LIN {X 0,Y 167.606,Z 477.864,A -85,B 0,C 180,E1 -23684.106,E2 -23684.106} C_VEL
LIN {X 0,Y 165.096,Z 487.968,A -85,B 0,C 180,E1 -23686.634,E2 -23686.634} C_VEL
LIN {X 0,Y 162.293,Z 498.184,A -85,B 0,C 180,E1 -23689.862,E2 -23689.862} C_VEL
LIN {X 0,Y 159.942,Z 506.695,A -85,B 0,C 180,E1 -23693.294,E2 -23693.294} C_VEL
LIN {X 0,Y 157.877,Z 514.165,A -85,B 0,C 180,E1 -23697.088,E2 -23697.088} C_VEL
LIN {X 0,Y 156.257,Z 520.604,A -85,B 0,C 180,E1 -23701.288,E2 -23701.288} C_VEL
LIN {X 0,Y 155.089,Z 526.085,A -85,B 0,C 180,E1 -23706.092,E2 -23706.092} C_VEL
LIN {X 0,Y 154.517,Z 529.018,A -85,B 0,C 180,E1 -23709.55,E2 -23709.55} C_VEL
LIN {X 0,Y 154.343,Z 531.312,A -85,B 0,C 180,E1 -23713.234,E2 -23713.234} C_VEL
LIN {X 0,Y 154.636,Z 532.81,A -85,B 0,C 180,E1 -23717.021,E2 -23717.021} C_VEL
LIN {X 0,Y 155.395,Z 533.466,A -85,B 0,C 180,E1 -23720.715,E2 -23720.715} C_VEL
LIN {X 0,Y 156.609,Z 533.371,A -85,B 0,C 180,E1 -23724.311,E2 -23724.311} C_VEL
LIN {X 0,Y 158.291,Z 532.569,A -85,B 0,C 180,E1 -23727.806,E2 -23727.806} C_VEL
LIN {X 0,Y 161.621,Z 529.982,A -85,B 0,C 180,E1 -23732.838,E2 -23732.838} C_VEL
LIN {X 0,Y 166.003,Z 525.79,A -85,B 0,C 180,E1 -23737.603,E2 -23737.603} C_VEL
LIN {X 0,Y 170.548,Z 520.782,A -85,B 0,C 180,E1 -23741.4,E2 -23741.4} C_VEL
LIN {X 0,Y 175.041,Z 515.343,A -85,B 0,C 180,E1 -23744.491,E2 -23744.491} C_VEL
LIN {X 0,Y 180.004,Z 508.62,A -85,B 0,C 180,E1 -23747.439,E2 -23747.439} C_VEL
LIN {X 0,Y 185.416,Z 500.371,A -85,B 0,C 180,E1 -23750.225,E2 -23750.225} C_VEL
LIN {X 0,Y 185.994,Z 499.153,A -85,B 0,C 180,E1 -23750.652,E2 -23750.652} C_VEL
LIN {X 0,Y 186.922,Z 493.836,A -85,B 0,C 180,E1 -23752.981,E2 -23752.981} C_VEL
LIN {X 0,Y 187.381,Z 487.918,A -85,B 0,C 180,E1 -23755.698,E2 -23755.698} C_VEL
LIN {X 0,Y 187.227,Z 483.523,A -85,B 0,C 180,E1 -23757.849,E2 -23757.849} C_VEL
LIN {X 0,Y 185.998,Z 477.859,A -85,B 0,C 180,E1 -23761.323,E2 -23761.323} C_VEL
LIN {X 0,Y 184.814,Z 473.591,A -85,B 0,C 180,E1 -23764.362,E2 -23764.362} C_VEL
LIN {X 0,Y 182.814,Z 469.179,A -85,B 0,C 180,E1 -23768.846,E2 -23768.846} C_VEL
LIN {X 0,Y 181.491,Z 465.804,A -85,B 0,C 180,E1 -23773.435,E2 -23773.435} C_VEL
LIN {X 0,Y 180.179,Z 465.166,A -85,B 0,C 180,E1 -23778.183,E2 -23778.183} C_VEL
LIN {X 0,Y 179.96,Z 465.653,A -85,B 0,C 180,E1 -23782.988,E2 -23782.988} C_VEL
LIN {X 0,Y 180.833,Z 467.315,A -85,B 0,C 180,E1 -23787.8,E2 -23787.8} C_VEL
LIN {X 0,Y 181.658,Z 470.723,A -85,B 0,C 180,E1 -23791.667,E2 -23791.667} C_VEL
LIN {X 0,Y 183.014,Z 474.33,A -85,B 0,C 180,E1 -23795.172,E2 -23795.172} C_VEL
LIN {X 0,Y 184.207,Z 478.675,A -85,B 0,C 180,E1 -23798.299,E2 -23798.299} C_VEL
LIN {X 0,Y 185.126,Z 482.365,A -85,B 0,C 180,E1 -23800.602,E2 -23800.602} C_VEL
LIN {X 0,Y 186.038,Z 487.75,A -85,B 0,C 180,E1 -23803.498,E2 -23803.498} C_VEL
LIN {X 0,Y 186.059,Z 492.37,A -85,B 0,C 180,E1 -23805.496,E2 -23805.496} C_VEL
LIN {X 0,Y 184.829,Z 499.849,A -85,B 0,C 180,E1 -23808.287,E2 -23808.287} C_VEL
LIN {X 0,Y 182.79,Z 507.719,A -85,B 0,C 180,E1 -23811.262,E2 -23811.262} C_VEL
LIN {X 0,Y 180.399,Z 513.668,A -85,B 0,C 180,E1 -23813.552,E2 -23813.552} C_VEL
LIN {X 0,Y 175.085,Z 521.477,A -85,B 0,C 180,E1 -23816.502,E2 -23816.502} C_VEL
LIN {X 0,Y 169.515,Z 528.822,A -85,B 0,C 180,E1 -23820.166,E2 -23820.166} C_VEL
LIN {X 0,Y 165.518,Z 533.839,A -85,B 0,C 180,E1 -23823.524,E2 -23823.524} C_VEL
LIN {X 0,Y 161.075,Z 538.896,A -85,B 0,C 180,E1 -23828.232,E2 -23828.232} C_VEL
LIN {X 0,Y 158.362,Z 541.598,A -85,B 0,C 180,E1 -23831.902,E2 -23831.902} C_VEL
LIN {X 0,Y 156.117,Z 543.873,A -85,B 0,C 180,E1 -23836.993,E2 -23836.993} C_VEL
LIN {X 0,Y 154.964,Z 544.594,A -85,B 0,C 180,E1 -23842.181,E2 -23842.181} C_VEL
LIN {X 0,Y 154.845,Z 543.82,A -85,B 0,C 180,E1 -23847.4,E2 -23847.4} C_VEL
LIN {X 0,Y 155.038,Z 542.857,A -85,B 0,C 180,E1 -23850.001,E2 -23850.001} C_VEL
LIN {X 0,Y 154.859,Z 541.002,A -85,B 0,C 180,E1 -23853.207,E2 -23853.207} C_VEL
LIN {X 0,Y 155.118,Z 537.201,A -85,B 0,C 180,E1 -23857.813,E2 -23857.813} C_VEL
LIN {X 0,Y 155.754,Z 532.742,A -85,B 0,C 180,E1 -23861.716,E2 -23861.716} C_VEL
LIN {X 0,Y 157.161,Z 525.927,A -85,B 0,C 180,E1 -23866.231,E2 -23866.231} C_VEL
LIN {X 0,Y 159.131,Z 518.527,A -85,B 0,C 180,E1 -23870.017,E2 -23870.017} C_VEL
LIN {X 0,Y 161.442,Z 509.83,A -85,B 0,C 180,E1 -23873.536,E2 -23873.536} C_VEL
LIN {X 0,Y 164.242,Z 499.771,A -85,B 0,C 180,E1 -23876.7,E2 -23876.7} C_VEL
LIN {X 0,Y 164.795,Z 496.433,A -85,B 0,C 180,E1 -23877.633,E2 -23877.633} C_VEL
LIN {X 0,Y 164.825,Z 485.619,A -85,B 0,C 180,E1 -23880.421,E2 -23880.421} C_VEL
LIN {X 0,Y 164.622,Z 480.666,A -85,B 0,C 180,E1 -23881.556,E2 -23881.556} C_VEL
LIN {X 0,Y 163.709,Z 475.807,A -85,B 0,C 180,E1 -23882.687,E2 -23882.687} C_VEL
LIN {X 0,Y 160.346,Z 468.173,A -85,B 0,C 180,E1 -23884.594,E2 -23884.594} C_VEL
LIN {X 0,Y 156.75,Z 460.325,A -85,B 0,C 180,E1 -23886.407,E2 -23886.407} C_VEL
LIN {X 0,Y 155.458,Z 455.118,A -85,B 0,C 180,E1 -23887.351,E2 -23887.351} C_VEL
LIN {X 0,Y 153.531,Z 445.023,A -85,B 0,C 180,E1 -23888.904,E2 -23888.904} C_VEL
LIN {X 0,Y 151.69,Z 438.84,A -85,B 0,C 180,E1 -23889.901,E2 -23889.901} C_VEL
LIN {X 0,Y 150.938,Z 435.132,A -85,B 0,C 180,E1 -23895.698,E2 -23895.698} C_VEL
LIN {X 0,Y 150.396,Z 431.753,A -85,B 0,C 180,E1 -23901.316,E2 -23901.316} C_VEL
LIN {X 0,Y 150.224,Z 431.776,A -85,B 0,C 180,E1 -23907.364,E2 -23907.364} C_VEL
LIN {X 0,Y 150.247,Z 431.754,A -85,B 0,C 180,E1 -23912.718,E2 -23912.718} C_VEL
LIN {X 0,Y 150.354,Z 431.756,A -85,B 0,C 180,E1 -23919.208,E2 -23919.208} C_VEL
LIN {X 0,Y 150.385,Z 431.751,A -85,B 0,C 180,E1 -23923.716,E2 -23923.716} C_VEL
LIN {X 0,Y 150.661,Z 431.712,A -85,B 0,C 180,E1 -23929.246,E2 -23929.246} C_VEL
LIN {X 0,Y 150.747,Z 431.705,A -85,B 0,C 180,E1 -23931.96,E2 -23931.96} C_VEL
LIN {X 0,Y 151.219,Z 431.645,A -85,B 0,C 180,E1 -23940,E2 -23940} C_VEL
LIN {X 0,Y 150.747,Z 431.703,A -85,B 0,C 180,E1 -23948.04,E2 -23948.04} C_VEL
LIN {X 0,Y 150.616,Z 431.717,A -85,B 0,C 180,E1 -23951.506,E2 -23951.506} C_VEL
LIN {X 0,Y 150.369,Z 431.724,A -85,B 0,C 180,E1 -23956.286,E2 -23956.286} C_VEL
LIN {X 0,Y 150.353,Z 431.734,A -85,B 0,C 180,E1 -23960.792,E2 -23960.792} C_VEL
LIN {X 0,Y 150.247,Z 431.769,A -85,B 0,C 180,E1 -23967.282,E2 -23967.282} C_VEL
LIN {X 0,Y 150.217,Z 431.757,A -85,B 0,C 180,E1 -23972.632,E2 -23972.632} C_VEL
LIN {X 0,Y 150.174,Z 431.754,A -85,B 0,C 180,E1 -23977.473,E2 -23977.473} C_VEL
LIN {X 0,Y 150.138,Z 431.779,A -85,B 0,C 180,E1 -23981.498,E2 -23981.498} C_VEL
LIN {X 0,Y 150.127,Z 431.782,A -85,B 0,C 180,E1 -23985.395,E2 -23985.395} C_VEL
LIN {X 0,Y 150.157,Z 431.764,A -85,B 0,C 180,E1 -23989.06,E2 -23989.06} C_VEL
LIN {X 0,Y 150.217,Z 431.756,A -85,B 0,C 180,E1 -23992.689,E2 -23992.689} C_VEL
LIN {X 0,Y 150.221,Z 431.772,A -85,B 0,C 180,E1 -23997.365,E2 -23997.365} C_VEL
LIN {X 0,Y 150.246,Z 431.755,A -85,B 0,C 180,E1 -24002.717,E2 -24002.717} C_VEL
LIN {X 0,Y 150.353,Z 431.755,A -85,B 0,C 180,E1 -24009.207,E2 -24009.207} C_VEL
LIN {X 0,Y 150.385,Z 431.75,A -85,B 0,C 180,E1 -24013.715,E2 -24013.715} C_VEL
LIN {X 0,Y 150.691,Z 431.709,A -85,B 0,C 180,E1 -24019.247,E2 -24019.247} C_VEL
LIN {X 0,Y 150.765,Z 431.706,A -85,B 0,C 180,E1 -24021.96,E2 -24021.96} C_VEL
LIN {X 0,Y 151.21,Z 431.654,A -85,B 0,C 180,E1 -24029.999,E2 -24029.999} C_VEL
LIN {X 0,Y 150.747,Z 431.7,A -85,B 0,C 180,E1 -24033.34,E2 -24033.34} C_VEL
LIN {X 0,Y 151.68,Z 434.542,A -85,B 0,C 180,E1 -24033.818,E2 -24033.818} C_VEL
LIN {X 0,Y 155.095,Z 443.394,A -85,B 0,C 180,E1 -24035.557,E2 -24035.557} C_VEL
LIN {X 0,Y 157.769,Z 455.58,A -85,B 0,C 180,E1 -24037.913,E2 -24037.913} C_VEL
LIN {X 0,Y 159.591,Z 466.873,A -85,B 0,C 180,E1 -24040.404,E2 -24040.404} C_VEL
LIN {X 0,Y 160.717,Z 477.996,A -85,B 0,C 180,E1 -24043.238,E2 -24043.238} C_VEL
LIN {X 0,Y 160.38,Z 480.569,A -85,B 0,C 180,E1 -24043.879,E2 -24043.879} C_VEL
LIN {X 0,Y 157.438,Z 491.337,A -85,B 0,C 180,E1 -24046.866,E2 -24046.866} C_VEL
LIN {X 0,Y 154.862,Z 500.222,A -85,B 0,C 180,E1 -24049.976,E2 -24049.976} C_VEL
LIN {X 0,Y 152.388,Z 508.801,A -85,B 0,C 180,E1 -24053.751,E2 -24053.751} C_VEL
LIN {X 0,Y 150.329,Z 516.089,A -85,B 0,C 180,E1 -24057.871,E2 -24057.871} C_VEL
LIN {X 0,Y 148.934,Z 521.626,A -85,B 0,C 180,E1 -24061.854,E2 -24061.854} C_VEL
LIN {X 0,Y 147.962,Z 526.248,A -85,B 0,C 180,E1 -24066.15,E2 -24066.15} C_VEL
LIN {X 0,Y 147.347,Z 529.542,A -85,B 0,C 180,E1 -24070.257,E2 -24070.257} C_VEL
LIN {X 0,Y 147.363,Z 532.428,A -85,B 0,C 180,E1 -24075.672,E2 -24075.672} C_VEL
LIN {X 0,Y 147.951,Z 533.48,A -85,B 0,C 180,E1 -24079.465,E2 -24079.465} C_VEL
LIN {X 0,Y 149.059,Z 533.812,A -85,B 0,C 180,E1 -24083.275,E2 -24083.275} C_VEL
LIN {X 0,Y 150.696,Z 533.398,A -85,B 0,C 180,E1 -24087.081,E2 -24087.081} C_VEL
LIN {X 0,Y 152.883,Z 532.17,A -85,B 0,C 180,E1 -24090.856,E2 -24090.856} C_VEL
LIN {X 0,Y 155.665,Z 530.091,A -85,B 0,C 180,E1 -24094.547,E2 -24094.547} C_VEL
LIN {X 0,Y 160.591,Z 525.711,A -85,B 0,C 180,E1 -24099.506,E2 -24099.506} C_VEL
LIN {X 0,Y 164.468,Z 521.812,A -85,B 0,C 180,E1 -24102.595,E2 -24102.595} C_VEL
LIN {X 0,Y 169.809,Z 515.754,A -85,B 0,C 180,E1 -24106.161,E2 -24106.161} C_VEL
LIN {X 0,Y 175.977,Z 507.825,A -85,B 0,C 180,E1 -24109.608,E2 -24109.608} C_VEL
LIN {X 0,Y 180.019,Z 502.001,A -85,B 0,C 180,E1 -24111.582,E2 -24111.582} C_VEL
LIN {X 0,Y 181.132,Z 498.231,A -85,B 0,C 180,E1 -24113.316,E2 -24113.316} C_VEL
LIN {X 0,Y 182.048,Z 491.436,A -85,B 0,C 180,E1 -24116.68,E2 -24116.68} C_VEL
LIN {X 0,Y 182.083,Z 487.42,A -85,B 0,C 180,E1 -24118.894,E2 -24118.894} C_VEL
LIN {X 0,Y 181.269,Z 482.422,A -85,B 0,C 180,E1 -24122.222,E2 -24122.222} C_VEL
LIN {X 0,Y 180.702,Z 479.514,A -85,B 0,C 180,E1 -24124.461,E2 -24124.461} C_VEL
LIN {X 0,Y 179.095,Z 475.199,A -85,B 0,C 180,E1 -24129.031,E2 -24129.031} C_VEL
LIN {X 0,Y 178.032,Z 471.992,A -85,B 0,C 180,E1 -24133.701,E2 -24133.701} C_VEL
LIN {X 0,Y 176.861,Z 471.49,A -85,B 0,C 180,E1 -24138.536,E2 -24138.536} C_VEL
LIN {X 0,Y 176.759,Z 472.209,A -85,B 0,C 180,E1 -24143.87,E2 -24143.87} C_VEL
LIN {X 0,Y 177.032,Z 472.822,A -85,B 0,C 180,E1 -24145.893,E2 -24145.893} C_VEL
LIN {X 0,Y 177.487,Z 474.141,A -85,B 0,C 180,E1 -24148.37,E2 -24148.37} C_VEL
LIN {X 0,Y 178.9,Z 479.645,A -85,B 0,C 180,E1 -24154.416,E2 -24154.416} C_VEL
LIN {X 0,Y 180.101,Z 485.351,A -85,B 0,C 180,E1 -24158.7,E2 -24158.7} C_VEL
LIN {X 0,Y 180.932,Z 491.56,A -85,B 0,C 180,E1 -24162.439,E2 -24162.439} C_VEL
LIN {X 0,Y 180.932,Z 494.505,A -85,B 0,C 180,E1 -24163.904,E2 -24163.904} C_VEL
LIN {X 0,Y 179.545,Z 501.474,A -85,B 0,C 180,E1 -24166.765,E2 -24166.765} C_VEL
LIN {X 0,Y 177.218,Z 509.076,A -85,B 0,C 180,E1 -24169.852,E2 -24169.852} C_VEL
LIN {X 0,Y 174.751,Z 514.717,A -85,B 0,C 180,E1 -24172.172,E2 -24172.172} C_VEL
LIN {X 0,Y 171.1,Z 519.894,A -85,B 0,C 180,E1 -24174.175,E2 -24174.175} C_VEL
LIN {X 0,Y 164.997,Z 527.506,A -85,B 0,C 180,E1 -24177.831,E2 -24177.831} C_VEL
LIN {X 0,Y 160.529,Z 532.689,A -85,B 0,C 180,E1 -24181.213,E2 -24181.213} C_VEL
LIN {X 0,Y 156.721,Z 536.813,A -85,B 0,C 180,E1 -24184.786,E2 -24184.786} C_VEL
LIN {X 0,Y 153.459,Z 539.994,A -85,B 0,C 180,E1 -24188.509,E2 -24188.509} C_VEL
LIN {X 0,Y 150.183,Z 542.867,A -85,B 0,C 180,E1 -24193.695,E2 -24193.695} C_VEL
LIN {X 0,Y 148.4,Z 544.179,A -85,B 0,C 180,E1 -24199.081,E2 -24199.081} C_VEL
LIN {X 0,Y 147.702,Z 544.023,A -85,B 0,C 180,E1 -24204.54,E2 -24204.54} C_VEL
LIN {X 0,Y 147.756,Z 543.383,A -85,B 0,C 180,E1 -24207.275,E2 -24207.275} C_VEL
LIN {X 0,Y 147.961,Z 542.311,A -85,B 0,C 180,E1 -24210.001,E2 -24210.001} C_VEL
LIN {X 0,Y 147.796,Z 540.593,A -85,B 0,C 180,E1 -24213.033,E2 -24213.033} C_VEL
LIN {X 0,Y 147.941,Z 537.676,A -85,B 0,C 180,E1 -24216.822,E2 -24216.822} C_VEL
LIN {X 0,Y 148.476,Z 533.464,A -85,B 0,C 180,E1 -24220.915,E2 -24220.915} C_VEL
LIN {X 0,Y 149.753,Z 527.028,A -85,B 0,C 180,E1 -24225.656,E2 -24225.656} C_VEL
LIN {X 0,Y 151.698,Z 519.972,A -85,B 0,C 180,E1 -24229.627,E2 -24229.627} C_VEL
LIN {X 0,Y 154.109,Z 511.148,A -85,B 0,C 180,E1 -24233.519,E2 -24233.519} C_VEL
LIN {X 0,Y 157.057,Z 501.178,A -85,B 0,C 180,E1 -24236.942,E2 -24236.942} C_VEL
LIN {X 0,Y 157.864,Z 498.001,A -85,B 0,C 180,E1 -24237.87,E2 -24237.87} C_VEL
LIN {X 0,Y 158.009,Z 487.611,A -85,B 0,C 180,E1 -24240.765,E2 -24240.765} C_VEL
LIN {X 0,Y 157.549,Z 475.881,A -85,B 0,C 180,E1 -24243.507,E2 -24243.507} C_VEL
LIN {X 0,Y 156.47,Z 462.878,A -85,B 0,C 180,E1 -24246.051,E2 -24246.051} C_VEL
LIN {X 0,Y 155.458,Z 455.118,A -85,B 0,C 180,E1 -24247.351,E2 -24247.351} C_VEL
LIN {X 0,Y 154.222,Z 451.815,A -85,B 0,C 180,E1 -24248.012,E2 -24248.012} C_VEL
LIN {X 0,Y 150.308,Z 447.483,A -85,B 0,C 180,E1 -24249.296,E2 -24249.296} C_VEL
LIN {X 0,Y 146.203,Z 443.152,A -85,B 0,C 180,E1 -24250.592,E2 -24250.592} C_VEL
LIN {X 0,Y 144.647,Z 439.82,A -85,B 0,C 180,E1 -24251.226,E2 -24251.226} C_VEL
LIN {X 0,Y 144.416,Z 438.578,A -85,B 0,C 180,E1 -24251.433,E2 -24251.433} C_VEL
LIN {X 0,Y 143.699,Z 435.125,A -85,B 0,C 180,E1 -24257.191,E2 -24257.191} C_VEL
LIN {X 0,Y 143.319,Z 432.633,A -85,B 0,C 180,E1 -24261.685,E2 -24261.685} C_VEL
LIN {X 0,Y 143.191,Z 432.651,A -85,B 0,C 180,E1 -24267.323,E2 -24267.323} C_VEL
LIN {X 0,Y 143.195,Z 432.634,A -85,B 0,C 180,E1 -24272.062,E2 -24272.062} C_VEL
LIN {X 0,Y 143.28,Z 432.639,A -85,B 0,C 180,E1 -24278.746,E2 -24278.746} C_VEL
LIN {X 0,Y 143.319,Z 432.629,A -85,B 0,C 180,E1 -24282.889,E2 -24282.889} C_VEL
LIN {X 0,Y 143.597,Z 432.591,A -85,B 0,C 180,E1 -24288.71,E2 -24288.71} C_VEL
LIN {X 0,Y 143.668,Z 432.588,A -85,B 0,C 180,E1 -24291.561,E2 -24291.561} C_VEL
LIN {X 0,Y 144.178,Z 432.522,A -85,B 0,C 180,E1 -24300,E2 -24300} C_VEL
LIN {X 0,Y 143.668,Z 432.586,A -85,B 0,C 180,E1 -24308.439,E2 -24308.439} C_VEL
LIN {X 0,Y 143.55,Z 432.597,A -85,B 0,C 180,E1 -24311.712,E2 -24311.712} C_VEL
LIN {X 0,Y 143.307,Z 432.597,A -85,B 0,C 180,E1 -24317.112,E2 -24317.112} C_VEL
LIN {X 0,Y 143.279,Z 432.617,A -85,B 0,C 180,E1 -24321.254,E2 -24321.254} C_VEL
LIN {X 0,Y 143.193,Z 432.647,A -85,B 0,C 180,E1 -24327.937,E2 -24327.937} C_VEL
LIN {X 0,Y 143.166,Z 432.631,A -85,B 0,C 180,E1 -24333.432,E2 -24333.432} C_VEL
LIN {X 0,Y 143.057,Z 432.655,A -85,B 0,C 180,E1 -24339.691,E2 -24339.691} C_VEL
LIN {X 0,Y 143.036,Z 432.666,A -85,B 0,C 180,E1 -24343.463,E2 -24343.463} C_VEL
LIN {X 0,Y 143.069,Z 432.655,A -85,B 0,C 180,E1 -24347.464,E2 -24347.464} C_VEL
LIN {X 0,Y 143.108,Z 432.637,A -85,B 0,C 180,E1 -24351.791,E2 -24351.791} C_VEL
LIN {X 0,Y 143.188,Z 432.648,A -85,B 0,C 180,E1 -24357.322,E2 -24357.322} C_VEL
LIN {X 0,Y 143.192,Z 432.635,A -85,B 0,C 180,E1 -24362.062,E2 -24362.062} C_VEL
LIN {X 0,Y 143.279,Z 432.637,A -85,B 0,C 180,E1 -24368.744,E2 -24368.744} C_VEL
LIN {X 0,Y 143.318,Z 432.627,A -85,B 0,C 180,E1 -24372.888,E2 -24372.888} C_VEL
LIN {X 0,Y 143.604,Z 432.592,A -85,B 0,C 180,E1 -24378.71,E2 -24378.71} C_VEL
LIN {X 0,Y 143.686,Z 432.587,A -85,B 0,C 180,E1 -24381.561,E2 -24381.561} C_VEL
LIN {X 0,Y 144.165,Z 432.531,A -85,B 0,C 180,E1 -24389.999,E2 -24389.999} C_VEL
LIN {X 0,Y 143.851,Z 432.562,A -85,B 0,C 180,E1 -24391.924,E2 -24391.924} C_VEL
LIN {X 0,Y 145.748,Z 437.9,A -85,B 0,C 180,E1 -24392.972,E2 -24392.972} C_VEL
LIN {X 0,Y 149.007,Z 446.478,A -85,B 0,C 180,E1 -24394.801,E2 -24394.801} C_VEL
LIN {X 0,Y 151.453,Z 458.476,A -85,B 0,C 180,E1 -24397.33,E2 -24397.33} C_VEL
LIN {X 0,Y 153.11,Z 470.258,A -85,B 0,C 180,E1 -24400.169,E2 -24400.169} C_VEL
LIN {X 0,Y 153.87,Z 480.076,A -85,B 0,C 180,E1 -24402.864,E2 -24402.864} C_VEL
LIN {X 0,Y 150.956,Z 490.342,A -85,B 0,C 180,E1 -24405.735,E2 -24405.735} C_VEL
LIN {X 0,Y 147.914,Z 500.569,A -85,B 0,C 180,E1 -24409.425,E2 -24409.425} C_VEL
LIN {X 0,Y 145.382,Z 508.987,A -85,B 0,C 180,E1 -24413.293,E2 -24413.293} C_VEL
LIN {X 0,Y 143.513,Z 515.375,A -85,B 0,C 180,E1 -24416.988,E2 -24416.988} C_VEL
LIN {X 0,Y 142.076,Z 520.933,A -85,B 0,C 180,E1 -24421.004,E2 -24421.004} C_VEL
LIN {X 0,Y 141.079,Z 525.25,A -85,B 0,C 180,E1 -24424.95,E2 -24424.95} C_VEL
LIN {X 0,Y 140.403,Z 528.463,A -85,B 0,C 180,E1 -24428.73,E2 -24428.73} C_VEL
LIN {X 0,Y 140.182,Z 530.173,A -85,B 0,C 180,E1 -24431.234,E2 -24431.234} C_VEL
LIN {X 0,Y 140.236,Z 532.319,A -85,B 0,C 180,E1 -24435.443,E2 -24435.443} C_VEL
LIN {X 0,Y 140.846,Z 533.611,A -85,B 0,C 180,E1 -24439.558,E2 -24439.558} C_VEL
LIN {X 0,Y 141.999,Z 534.126,A -85,B 0,C 180,E1 -24443.565,E2 -24443.565} C_VEL
LIN {X 0,Y 143.654,Z 533.853,A -85,B 0,C 180,E1 -24447.442,E2 -24447.442} C_VEL
LIN {X 0,Y 145.807,Z 532.885,A -85,B 0,C 180,E1 -24451.183,E2 -24451.183} C_VEL
LIN {X 0,Y 149.992,Z 530.143,A -85,B 0,C 180,E1 -24456.531,E2 -24456.531} C_VEL
LIN {X 0,Y 155.476,Z 525.543,A -85,B 0,C 180,E1 -24461.666,E2 -24461.666} C_VEL
LIN {X 0,Y 161.117,Z 520.115,A -85,B 0,C 180,E1 -24465.693,E2 -24465.693} C_VEL
LIN {X 0,Y 167.273,Z 513.308,A -85,B 0,C 180,E1 -24469.328,E2 -24469.328} C_VEL
LIN {X 0,Y 173.825,Z 504.974,A -85,B 0,C 180,E1 -24472.597,E2 -24472.597} C_VEL
LIN {X 0,Y 174.701,Z 503.68,A -85,B 0,C 180,E1 -24473.068,E2 -24473.068} C_VEL
LIN {X 0,Y 175.951,Z 499.129,A -85,B 0,C 180,E1 -24475.418,E2 -24475.418} C_VEL
LIN {X 0,Y 176.722,Z 494.898,A -85,B 0,C 180,E1 -24477.721,E2 -24477.721} C_VEL
LIN {X 0,Y 176.899,Z 491.184,A -85,B 0,C 180,E1 -24480,E2 -24480} C_VEL
LIN {X 0,Y 176.439,Z 486.58,A -85,B 0,C 180,E1 -24483.426,E2 -24483.426} C_VEL
LIN {X 0,Y 175.934,Z 484.022,A -85,B 0,C 180,E1 -24485.732,E2 -24485.732} C_VEL
LIN {X 0,Y 175.056,Z 481.008,A -85,B 0,C 180,E1 -24489.241,E2 -24489.241} C_VEL
LIN {X 0,Y 174.117,Z 477.936,A -85,B 0,C 180,E1 -24494.372,E2 -24494.372} C_VEL
LIN {X 0,Y 173.055,Z 477.751,A -85,B 0,C 180,E1 -24500.927,E2 -24500.927} C_VEL
LIN {X 0,Y 173.161,Z 478.355,A -85,B 0,C 180,E1 -24503.946,E2 -24503.946} C_VEL
LIN {X 0,Y 173.494,Z 479.509,A -85,B 0,C 180,E1 -24506.98,E2 -24506.98} C_VEL
LIN {X 0,Y 173.848,Z 481.766,A -85,B 0,C 180,E1 -24510.209,E2 -24510.209} C_VEL
LIN {X 0,Y 174.675,Z 485.537,A -85,B 0,C 180,E1 -24514.284,E2 -24514.284} C_VEL
LIN {X 0,Y 175.348,Z 490.022,A -85,B 0,C 180,E1 -24517.874,E2 -24517.874} C_VEL
LIN {X 0,Y 175.754,Z 495.166,A -85,B 0,C 180,E1 -24521.283,E2 -24521.283} C_VEL
LIN {X 0,Y 175.566,Z 498.618,A -85,B 0,C 180,E1 -24523.148,E2 -24523.148} C_VEL
LIN {X 0,Y 173.888,Z 504.629,A -85,B 0,C 180,E1 -24525.814,E2 -24525.814} C_VEL
LIN {X 0,Y 171.214,Z 511.821,A -85,B 0,C 180,E1 -24528.948,E2 -24528.948} C_VEL
LIN {X 0,Y 168.416,Z 517.048,A -85,B 0,C 180,E1 -24531.249,E2 -24531.249} C_VEL
LIN {X 0,Y 162.646,Z 524.098,A -85,B 0,C 180,E1 -24534.316,E2 -24534.316} C_VEL
LIN {X 0,Y 157.393,Z 529.889,A -85,B 0,C 180,E1 -24537.601,E2 -24537.601} C_VEL
LIN {X 0,Y 153.566,Z 533.91,A -85,B 0,C 180,E1 -24540.622,E2 -24540.622} C_VEL
LIN {X 0,Y 149.094,Z 538.173,A -85,B 0,C 180,E1 -24544.899,E2 -24544.899} C_VEL
LIN {X 0,Y 144.922,Z 541.632,A -85,B 0,C 180,E1 -24550.157,E2 -24550.157} C_VEL
LIN {X 0,Y 142.241,Z 543.529,A -85,B 0,C 180,E1 -24555.698,E2 -24555.698} C_VEL
LIN {X 0,Y 140.895,Z 543.974,A -85,B 0,C 180,E1 -24561.395,E2 -24561.395} C_VEL
LIN {X 0,Y 140.629,Z 543.635,A -85,B 0,C 180,E1 -24564.265,E2 -24564.265} C_VEL
LIN {X 0,Y 140.705,Z 542.799,A -85,B 0,C 180,E1 -24567.404,E2 -24567.404} C_VEL
LIN {X 0,Y 140.885,Z 541.758,A -85,B 0,C 180,E1 -24570.001,E2 -24570.001} C_VEL
LIN {X 0,Y 140.71,Z 539.197,A -85,B 0,C 180,E1 -24574.298,E2 -24574.298} C_VEL
LIN {X 0,Y 141.02,Z 535.594,A -85,B 0,C 180,E1 -24578.6,E2 -24578.6} C_VEL
LIN {X 0,Y 141.801,Z 530.841,A -85,B 0,C 180,E1 -24582.888,E2 -24582.888} C_VEL
LIN {X 0,Y 143.558,Z 523.697,A -85,B 0,C 180,E1 -24587.818,E2 -24587.818} C_VEL
LIN {X 0,Y 145.781,Z 515.862,A -85,B 0,C 180,E1 -24591.94,E2 -24591.94} C_VEL
LIN {X 0,Y 148.425,Z 506.879,A -85,B 0,C 180,E1 -24595.653,E2 -24595.653} C_VEL
LIN {X 0,Y 150.942,Z 498.204,A -85,B 0,C 180,E1 -24598.507,E2 -24598.507} C_VEL
LIN {X 0,Y 151.165,Z 487.348,A -85,B 0,C 180,E1 -24601.694,E2 -24601.694} C_VEL
LIN {X 0,Y 150.717,Z 475.232,A -85,B 0,C 180,E1 -24604.665,E2 -24604.665} C_VEL
LIN {X 0,Y 149.806,Z 463.418,A -85,B 0,C 180,E1 -24607.104,E2 -24607.104} C_VEL
LIN {X 0,Y 148.41,Z 452.659,A -85,B 0,C 180,E1 -24609.006,E2 -24609.006} C_VEL
LIN {X 0,Y 146.736,Z 445.408,A -85,B 0,C 180,E1 -24610.22,E2 -24610.22} C_VEL
LIN {X 0,Y 144.647,Z 439.82,A -85,B 0,C 180,E1 -24611.226,E2 -24611.226} C_VEL
LIN {X 0,Y 143.994,Z 438.659,A -85,B 0,C 180,E1 -24611.666,E2 -24611.666} C_VEL
LIN {X 0,Y 139.348,Z 436.334,A -85,B 0,C 180,E1 -24616.076,E2 -24616.076} C_VEL
LIN {X 0,Y 137.078,Z 434.785,A -85,B 0,C 180,E1 -24619.668,E2 -24619.668} C_VEL
LIN {X 0,Y 136.227,Z 433.622,A -85,B 0,C 180,E1 -24622.453,E2 -24622.453} C_VEL
LIN {X 0,Y 136.144,Z 433.515,A -85,B 0,C 180,E1 -24623.403,E2 -24623.403} C_VEL
LIN {X 0,Y 136.07,Z 433.538,A -85,B 0,C 180,E1 -24628.902,E2 -24628.902} C_VEL
LIN {X 0,Y 136.15,Z 433.509,A -85,B 0,C 180,E1 -24632.317,E2 -24632.317} C_VEL
LIN {X 0,Y 136.246,Z 433.515,A -85,B 0,C 180,E1 -24638.833,E2 -24638.833} C_VEL
LIN {X 0,Y 136.287,Z 433.51,A -85,B 0,C 180,E1 -24645.058,E2 -24645.058} C_VEL
LIN {X 0,Y 136.5,Z 433.475,A -85,B 0,C 180,E1 -24648.115,E2 -24648.115} C_VEL
LIN {X 0,Y 136.595,Z 433.468,A -85,B 0,C 180,E1 -24651.12,E2 -24651.12} C_VEL
LIN {X 0,Y 137.135,Z 433.399,A -85,B 0,C 180,E1 -24660,E2 -24660} C_VEL
LIN {X 0,Y 136.594,Z 433.469,A -85,B 0,C 180,E1 -24668.879,E2 -24668.879} C_VEL
LIN {X 0,Y 136.494,Z 433.476,A -85,B 0,C 180,E1 -24671.954,E2 -24671.954} C_VEL
LIN {X 0,Y 136.246,Z 433.473,A -85,B 0,C 180,E1 -24678.029,E2 -24678.029} C_VEL
LIN {X 0,Y 136.2,Z 433.502,A -85,B 0,C 180,E1 -24681.748,E2 -24681.748} C_VEL
LIN {X 0,Y 136.118,Z 433.529,A -85,B 0,C 180,E1 -24688.628,E2 -24688.628} C_VEL
LIN {X 0,Y 136.072,Z 433.502,A -85,B 0,C 180,E1 -24694.62,E2 -24694.62} C_VEL
LIN {X 0,Y 136.029,Z 433.525,A -85,B 0,C 180,E1 -24699.195,E2 -24699.195} C_VEL
LIN {X 0,Y 135.981,Z 433.545,A -85,B 0,C 180,E1 -24703.649,E2 -24703.649} C_VEL
LIN {X 0,Y 136.033,Z 433.53,A -85,B 0,C 180,E1 -24707.806,E2 -24707.806} C_VEL
LIN {X 0,Y 136.057,Z 433.513,A -85,B 0,C 180,E1 -24711.693,E2 -24711.693} C_VEL
LIN {X 0,Y 136.092,Z 433.53,A -85,B 0,C 180,E1 -24715.717,E2 -24715.717} C_VEL
LIN {X 0,Y 136.148,Z 433.511,A -85,B 0,C 180,E1 -24722.316,E2 -24722.316} C_VEL
LIN {X 0,Y 136.246,Z 433.513,A -85,B 0,C 180,E1 -24728.832,E2 -24728.832} C_VEL
LIN {X 0,Y 136.287,Z 433.511,A -85,B 0,C 180,E1 -24735.057,E2 -24735.057} C_VEL
LIN {X 0,Y 136.503,Z 433.477,A -85,B 0,C 180,E1 -24738.114,E2 -24738.114} C_VEL
LIN {X 0,Y 136.61,Z 433.469,A -85,B 0,C 180,E1 -24741.121,E2 -24741.121} C_VEL
LIN {X 0,Y 137.122,Z 433.409,A -85,B 0,C 180,E1 -24749.999,E2 -24749.999} C_VEL
LIN {X 0,Y 137.045,Z 433.418,A -85,B 0,C 180,E1 -24750.367,E2 -24750.367} C_VEL
LIN {X 0,Y 138.047,Z 436.411,A -85,B 0,C 180,E1 -24751.003,E2 -24751.003} C_VEL
LIN {X 0,Y 142.552,Z 448.259,A -85,B 0,C 180,E1 -24753.763,E2 -24753.763} C_VEL
LIN {X 0,Y 144.792,Z 459.326,A -85,B 0,C 180,E1 -24756.269,E2 -24756.269} C_VEL
LIN {X 0,Y 146.407,Z 471.358,A -85,B 0,C 180,E1 -24759.323,E2 -24759.323} C_VEL
LIN {X 0,Y 147.066,Z 480.809,A -85,B 0,C 180,E1 -24762.067,E2 -24762.067} C_VEL
LIN {X 0,Y 143.966,Z 491.297,A -85,B 0,C 180,E1 -24765.174,E2 -24765.174} C_VEL
LIN {X 0,Y 141.025,Z 500.751,A -85,B 0,C 180,E1 -24768.761,E2 -24768.761} C_VEL
LIN {X 0,Y 138.322,Z 509.418,A -85,B 0,C 180,E1 -24772.948,E2 -24772.948} C_VEL
LIN {X 0,Y 136.066,Z 516.981,A -85,B 0,C 180,E1 -24777.7,E2 -24777.7} C_VEL
LIN {X 0,Y 134.339,Z 523.608,A -85,B 0,C 180,E1 -24783.171,E2 -24783.171} C_VEL
LIN {X 0,Y 133.417,Z 527.778,A -85,B 0,C 180,E1 -24787.8,E2 -24787.8} C_VEL
LIN {X 0,Y 133.044,Z 531.329,A -85,B 0,C 180,E1 -24793.369,E2 -24793.369} C_VEL
LIN {X 0,Y 133.359,Z 533.113,A -85,B 0,C 180,E1 -24797.542,E2 -24797.542} C_VEL
LIN {X 0,Y 134.255,Z 534.13,A -85,B 0,C 180,E1 -24801.739,E2 -24801.739} C_VEL
LIN {X 0,Y 135.74,Z 534.402,A -85,B 0,C 180,E1 -24805.933,E2 -24805.933} C_VEL
LIN {X 0,Y 137.839,Z 533.931,A -85,B 0,C 180,E1 -24810.083,E2 -24810.083} C_VEL
LIN {X 0,Y 140.563,Z 532.679,A -85,B 0,C 180,E1 -24814.152,E2 -24814.152} C_VEL
LIN {X 0,Y 143.947,Z 530.572,A -85,B 0,C 180,E1 -24818.067,E2 -24818.067} C_VEL
LIN {X 0,Y 147.951,Z 527.601,A -85,B 0,C 180,E1 -24821.809,E2 -24821.809} C_VEL
LIN {X 0,Y 153.739,Z 522.715,A -85,B 0,C 180,E1 -24826.103,E2 -24826.103} C_VEL
LIN {X 0,Y 159.993,Z 516.551,A -85,B 0,C 180,E1 -24829.88,E2 -24829.88} C_VEL
LIN {X 0,Y 166.899,Z 508.719,A -85,B 0,C 180,E1 -24833.351,E2 -24833.351} C_VEL
LIN {X 0,Y 168.394,Z 506.882,A -85,B 0,C 180,E1 -24834.012,E2 -24834.012} C_VEL
LIN {X 0,Y 169.387,Z 505.266,A -85,B 0,C 180,E1 -24834.718,E2 -24834.718} C_VEL
LIN {X 0,Y 170.945,Z 500.248,A -85,B 0,C 180,E1 -24837.644,E2 -24837.644} C_VEL
LIN {X 0,Y 171.61,Z 496.497,A -85,B 0,C 180,E1 -24840,E2 -24840} C_VEL
LIN {X 0,Y 171.589,Z 491.75,A -85,B 0,C 180,E1 -24843.732,E2 -24843.732} C_VEL
LIN {X 0,Y 171.115,Z 488.454,A -85,B 0,C 180,E1 -24847.078,E2 -24847.078} C_VEL
LIN {X 0,Y 170.705,Z 486.598,A -85,B 0,C 180,E1 -24849.479,E2 -24849.479} C_VEL
LIN {X 0,Y 170.133,Z 483.811,A -85,B 0,C 180,E1 -24854.351,E2 -24854.351} C_VEL
LIN {X 0,Y 169.23,Z 483.57,A -85,B 0,C 180,E1 -24859.405,E2 -24859.405} C_VEL
LIN {X 0,Y 169.221,Z 484.483,A -85,B 0,C 180,E1 -24864.539,E2 -24864.539} C_VEL
LIN {X 0,Y 169.465,Z 485.541,A -85,B 0,C 180,E1 -24867.142,E2 -24867.142} C_VEL
LIN {X 0,Y 169.757,Z 488.466,A -85,B 0,C 180,E1 -24871.165,E2 -24871.165} C_VEL
LIN {X 0,Y 170.009,Z 489.533,A -85,B 0,C 180,E1 -24872.507,E2 -24872.507} C_VEL
LIN {X 0,Y 170.429,Z 494.088,A -85,B 0,C 180,E1 -24876.69,E2 -24876.69} C_VEL
LIN {X 0,Y 170.551,Z 498.158,A -85,B 0,C 180,E1 -24879.695,E2 -24879.695} C_VEL
LIN {X 0,Y 170.247,Z 501.844,A -85,B 0,C 180,E1 -24882.009,E2 -24882.009} C_VEL
LIN {X 0,Y 168.259,Z 507.637,A -85,B 0,C 180,E1 -24884.761,E2 -24884.761} C_VEL
LIN {X 0,Y 165.233,Z 514.333,A -85,B 0,C 180,E1 -24887.942,E2 -24887.942} C_VEL
LIN {X 0,Y 162.983,Z 518.085,A -85,B 0,C 180,E1 -24889.7,E2 -24889.7} C_VEL
LIN {X 0,Y 156.981,Z 524.882,A -85,B 0,C 180,E1 -24892.816,E2 -24892.816} C_VEL
LIN {X 0,Y 151.483,Z 530.434,A -85,B 0,C 180,E1 -24896.171,E2 -24896.171} C_VEL
LIN {X 0,Y 145.341,Z 536.139,A -85,B 0,C 180,E1 -24901.084,E2 -24901.084} C_VEL
LIN {X 0,Y 142.678,Z 538.382,A -85,B 0,C 180,E1 -24903.685,E2 -24903.685} C_VEL
LIN {X 0,Y 138.24,Z 541.612,A -85,B 0,C 180,E1 -24909.154,E2 -24909.154} C_VEL
LIN {X 0,Y 135.347,Z 543.354,A -85,B 0,C 180,E1 -24914.953,E2 -24914.953} C_VEL
LIN {X 0,Y 133.858,Z 543.634,A -85,B 0,C 180,E1 -24920.939,E2 -24920.939} C_VEL
LIN {X 0,Y 133.596,Z 542.377,A -85,B 0,C 180,E1 -24926.986,E2 -24926.986} C_VEL
LIN {X 0,Y 133.811,Z 541.178,A -85,B 0,C 180,E1 -24930.001,E2 -24930.001} C_VEL
LIN {X 0,Y 133.65,Z 538.486,A -85,B 0,C 180,E1 -24934.525,E2 -24934.525} C_VEL
LIN {X 0,Y 134.006,Z 534.751,A -85,B 0,C 180,E1 -24939.053,E2 -24939.053} C_VEL
LIN {X 0,Y 134.846,Z 529.853,A -85,B 0,C 180,E1 -24943.565,E2 -24943.565} C_VEL
LIN {X 0,Y 136.422,Z 523.674,A -85,B 0,C 180,E1 -24948.006,E2 -24948.006} C_VEL
LIN {X 0,Y 138.745,Z 515.928,A -85,B 0,C 180,E1 -24952.329,E2 -24952.329} C_VEL
LIN {X 0,Y 141.7,Z 506.25,A -85,B 0,C 180,E1 -24956.513,E2 -24956.513} C_VEL
LIN {X 0,Y 144.043,Z 498.408,A -85,B 0,C 180,E1 -24959.204,E2 -24959.204} C_VEL
LIN {X 0,Y 144.354,Z 488.232,A -85,B 0,C 180,E1 -24962.382,E2 -24962.382} C_VEL
LIN {X 0,Y 144.099,Z 477.404,A -85,B 0,C 180,E1 -24965.254,E2 -24965.254} C_VEL
LIN {X 0,Y 143.356,Z 465.57,A -85,B 0,C 180,E1 -24967.881,E2 -24967.881} C_VEL
LIN {X 0,Y 141.859,Z 453.282,A -85,B 0,C 180,E1 -24970.222,E2 -24970.222} C_VEL
LIN {X 0,Y 139.809,Z 445.598,A -85,B 0,C 180,E1 -24971.694,E2 -24971.694} C_VEL
LIN {X 0,Y 137.343,Z 439.216,A -85,B 0,C 180,E1 -24972.966,E2 -24972.966} C_VEL
LIN {X 0,Y 137.153,Z 438.3,A -85,B 0,C 180,E1 -24973.168,E2 -24973.168} C_VEL
LIN {X 0,Y 136.425,Z 434.124,A -85,B 0,C 180,E1 -24980.601,E2 -24980.601} C_VEL
LIN {X 0,Y 136.219,Z 433.514,A -85,B 0,C 180,E1 -24982.217,E2 -24982.217} C_VEL
LIN {X 0,Y 136.144,Z 433.515,A -85,B 0,C 180,E1 -24983.403,E2 -24983.403} C_VEL
LIN {X 0,Y 135.409,Z 433.615,A -85,B 0,C 180,E1 -24985.87,E2 -24985.87} C_VEL
LIN {X 0,Y 133.773,Z 433.824,A -85,B 0,C 180,E1 -24988.301,E2 -24988.301} C_VEL
LIN {X 0,Y 129.278,Z 434.371,A -85,B 0,C 180,E1 -24995.02,E2 -24995.02} C_VEL
LIN {X 0,Y 129.051,Z 434.402,A -85,B 0,C 180,E1 -24996.796,E2 -24996.796} C_VEL
LIN {X 0,Y 129.162,Z 434.391,A -85,B 0,C 180,E1 -25000.945,E2 -25000.945} C_VEL
LIN {X 0,Y 129.419,Z 434.357,A -85,B 0,C 180,E1 -25007.82,E2 -25007.82} C_VEL
LIN {X 0,Y 129.52,Z 434.347,A -85,B 0,C 180,E1 -25010.631,E2 -25010.631} C_VEL
LIN {X 0,Y 130.091,Z 434.277,A -85,B 0,C 180,E1 -25020,E2 -25020} C_VEL
LIN {X 0,Y 129.52,Z 434.348,A -85,B 0,C 180,E1 -25029.368,E2 -25029.368} C_VEL
LIN {X 0,Y 129.395,Z 434.357,A -85,B 0,C 180,E1 -25032.548,E2 -25032.548} C_VEL
LIN {X 0,Y 129.156,Z 434.358,A -85,B 0,C 180,E1 -25039.056,E2 -25039.056} C_VEL
LIN {X 0,Y 129.111,Z 434.388,A -85,B 0,C 180,E1 -25042.398,E2 -25042.398} C_VEL
LIN {X 0,Y 129.038,Z 434.408,A -85,B 0,C 180,E1 -25049.373,E2 -25049.373} C_VEL
LIN {X 0,Y 128.981,Z 434.382,A -85,B 0,C 180,E1 -25055.18,E2 -25055.18} C_VEL
LIN {X 0,Y 128.925,Z 434.418,A -85,B 0,C 180,E1 -25060.855,E2 -25060.855} C_VEL
LIN {X 0,Y 128.919,Z 434.424,A -85,B 0,C 180,E1 -25065.128,E2 -25065.128} C_VEL
LIN {X 0,Y 128.958,Z 434.398,A -85,B 0,C 180,E1 -25069.727,E2 -25069.727} C_VEL
LIN {X 0,Y 128.994,Z 434.41,A -85,B 0,C 180,E1 -25074.81,E2 -25074.81} C_VEL
LIN {X 0,Y 129.053,Z 434.401,A -85,B 0,C 180,E1 -25080.65,E2 -25080.65} C_VEL
LIN {X 0,Y 129.109,Z 434.403,A -85,B 0,C 180,E1 -25087.727,E2 -25087.727} C_VEL
LIN {X 0,Y 129.162,Z 434.387,A -85,B 0,C 180,E1 -25090.944,E2 -25090.944} C_VEL
LIN {X 0,Y 129.42,Z 434.361,A -85,B 0,C 180,E1 -25097.814,E2 -25097.814} C_VEL
LIN {X 0,Y 129.532,Z 434.349,A -85,B 0,C 180,E1 -25100.631,E2 -25100.631} C_VEL
LIN {X 0,Y 129.877,Z 434.304,A -85,B 0,C 180,E1 -25108.642,E2 -25108.642} C_VEL
LIN {X 0,Y 130.996,Z 437.189,A -85,B 0,C 180,E1 -25109.326,E2 -25109.326} C_VEL
LIN {X 0,Y 134.891,Z 446.81,A -85,B 0,C 180,E1 -25111.753,E2 -25111.753} C_VEL
LIN {X 0,Y 136.783,Z 452.734,A -85,B 0,C 180,E1 -25113.27,E2 -25113.27} C_VEL
LIN {X 0,Y 138.752,Z 464.284,A -85,B 0,C 180,E1 -25116.178,E2 -25116.178} C_VEL
LIN {X 0,Y 139.952,Z 475.628,A -85,B 0,C 180,E1 -25119.392,E2 -25119.392} C_VEL
LIN {X 0,Y 140.285,Z 481.375,A -85,B 0,C 180,E1 -25121.193,E2 -25121.193} C_VEL
LIN {X 0,Y 137.211,Z 491.369,A -85,B 0,C 180,E1 -25124.289,E2 -25124.289} C_VEL
LIN {X 0,Y 133.892,Z 501.575,A -85,B 0,C 180,E1 -25128.356,E2 -25128.356} C_VEL
LIN {X 0,Y 131.095,Z 510.306,A -85,B 0,C 180,E1 -25132.877,E2 -25132.877} C_VEL
LIN {X 0,Y 128.712,Z 518.015,A -85,B 0,C 180,E1 -25138.085,E2 -25138.085} C_VEL
LIN {X 0,Y 127.125,Z 524.146,A -85,B 0,C 180,E1 -25143.56,E2 -25143.56} C_VEL
LIN {X 0,Y 126.176,Z 528.462,A -85,B 0,C 180,E1 -25148.758,E2 -25148.758} C_VEL
LIN {X 0,Y 125.945,Z 531.341,A -85,B 0,C 180,E1 -25153.496,E2 -25153.496} C_VEL
LIN {X 0,Y 126.346,Z 533.282,A -85,B 0,C 180,E1 -25158.126,E2 -25158.126} C_VEL
LIN {X 0,Y 127.367,Z 534.368,A -85,B 0,C 180,E1 -25162.629,E2 -25162.629} C_VEL
LIN {X 0,Y 128.995,Z 534.709,A -85,B 0,C 180,E1 -25166.987,E2 -25166.987} C_VEL
LIN {X 0,Y 131.204,Z 534.347,A -85,B 0,C 180,E1 -25171.178,E2 -25171.178} C_VEL
LIN {X 0,Y 133.923,Z 533.248,A -85,B 0,C 180,E1 -25175.177,E2 -25175.177} C_VEL
LIN {X 0,Y 137.263,Z 531.468,A -85,B 0,C 180,E1 -25178.998,E2 -25178.998} C_VEL
LIN {X 0,Y 143.217,Z 527.504,A -85,B 0,C 180,E1 -25184.272,E2 -25184.272} C_VEL
LIN {X 0,Y 148.059,Z 523.673,A -85,B 0,C 180,E1 -25187.668,E2 -25187.668} C_VEL
LIN {X 0,Y 154.627,Z 517.751,A -85,B 0,C 180,E1 -25191.506,E2 -25191.506} C_VEL
LIN {X 0,Y 161.869,Z 510.16,A -85,B 0,C 180,E1 -25195.019,E2 -25195.019} C_VEL
LIN {X 0,Y 163.534,Z 508.232,A -85,B 0,C 180,E1 -25195.789,E2 -25195.789} C_VEL
LIN {X 0,Y 164.839,Z 505.29,A -85,B 0,C 180,E1 -25197.557,E2 -25197.557} C_VEL
LIN {X 0,Y 165.969,Z 501.586,A -85,B 0,C 180,E1 -25200,E2 -25200} C_VEL
LIN {X 0,Y 166.415,Z 498.523,A -85,B 0,C 180,E1 -25202.421,E2 -25202.421} C_VEL
LIN {X 0,Y 166.487,Z 494.698,A -85,B 0,C 180,E1 -25206.058,E2 -25206.058} C_VEL
LIN {X 0,Y 166.096,Z 491.952,A -85,B 0,C 180,E1 -25209.745,E2 -25209.745} C_VEL
LIN {X 0,Y 165.739,Z 489.431,A -85,B 0,C 180,E1 -25214.74,E2 -25214.74} C_VEL
LIN {X 0,Y 164.913,Z 489.366,A -85,B 0,C 180,E1 -25220.358,E2 -25220.358} C_VEL
LIN {X 0,Y 164.959,Z 490.455,A -85,B 0,C 180,E1 -25225.217,E2 -25225.217} C_VEL
LIN {X 0,Y 165.106,Z 491.772,A -85,B 0,C 180,E1 -25227.92,E2 -25227.92} C_VEL
LIN {X 0,Y 165.273,Z 494.469,A -85,B 0,C 180,E1 -25231.739,E2 -25231.739} C_VEL
LIN {X 0,Y 165.396,Z 496.932,A -85,B 0,C 180,E1 -25234.353,E2 -25234.353} C_VEL
LIN {X 0,Y 165.348,Z 500.537,A -85,B 0,C 180,E1 -25237.544,E2 -25237.544} C_VEL
LIN {X 0,Y 165.118,Z 503.768,A -85,B 0,C 180,E1 -25239.993,E2 -25239.993} C_VEL
LIN {X 0,Y 164.834,Z 505.185,A -85,B 0,C 180,E1 -25240.914,E2 -25240.914} C_VEL
LIN {X 0,Y 162.478,Z 510.791,A -85,B 0,C 180,E1 -25243.795,E2 -25243.795} C_VEL
LIN {X 0,Y 159.248,Z 516.719,A -85,B 0,C 180,E1 -25246.841,E2 -25246.841} C_VEL
LIN {X 0,Y 156.648,Z 520.231,A -85,B 0,C 180,E1 -25248.568,E2 -25248.568} C_VEL
LIN {X 0,Y 149.402,Z 527.53,A -85,B 0,C 180,E1 -25252.301,E2 -25252.301} C_VEL
LIN {X 0,Y 143.906,Z 532.513,A -85,B 0,C 180,E1 -25255.833,E2 -25255.833} C_VEL
LIN {X 0,Y 137.721,Z 537.537,A -85,B 0,C 180,E1 -25261.003,E2 -25261.003} C_VEL
LIN {X 0,Y 133.854,Z 540.252,A -85,B 0,C 180,E1 -25265.164,E2 -25265.164} C_VEL
LIN {X 0,Y 129.781,Z 542.568,A -85,B 0,C 180,E1 -25271.041,E2 -25271.041} C_VEL
LIN {X 0,Y 127.475,Z 543.394,A -85,B 0,C 180,E1 -25277.261,E2 -25277.261} C_VEL
LIN {X 0,Y 126.52,Z 542.743,A -85,B 0,C 180,E1 -25283.623,E2 -25283.623} C_VEL
LIN {X 0,Y 126.587,Z 541.461,A -85,B 0,C 180,E1 -25287.929,E2 -25287.929} C_VEL
LIN {X 0,Y 126.742,Z 540.589,A -85,B 0,C 180,E1 -25290.001,E2 -25290.001} C_VEL
LIN {X 0,Y 126.598,Z 537.762,A -85,B 0,C 180,E1 -25294.778,E2 -25294.778} C_VEL
LIN {X 0,Y 126.987,Z 533.871,A -85,B 0,C 180,E1 -25299.558,E2 -25299.558} C_VEL
LIN {X 0,Y 127.925,Z 528.803,A -85,B 0,C 180,E1 -25304.314,E2 -25304.314} C_VEL
LIN {X 0,Y 129.685,Z 522.403,A -85,B 0,C 180,E1 -25308.976,E2 -25308.976} C_VEL
LIN {X 0,Y 132.172,Z 514.424,A -85,B 0,C 180,E1 -25313.504,E2 -25313.504} C_VEL
LIN {X 0,Y 134.761,Z 506.291,A -85,B 0,C 180,E1 -25317.151,E2 -25317.151} C_VEL
LIN {X 0,Y 137.157,Z 498.52,A -85,B 0,C 180,E1 -25319.973,E2 -25319.973} C_VEL
LIN {X 0,Y 137.539,Z 488.347,A -85,B 0,C 180,E1 -25323.32,E2 -25323.32} C_VEL
LIN {X 0,Y 137.406,Z 478.084,A -85,B 0,C 180,E1 -25326.206,E2 -25326.206} C_VEL
LIN {X 0,Y 136.74,Z 465.927,A -85,B 0,C 180,E1 -25329.1,E2 -25329.1} C_VEL
LIN {X 0,Y 135.598,Z 455.366,A -85,B 0,C 180,E1 -25331.276,E2 -25331.276} C_VEL
LIN {X 0,Y 133.722,Z 448.48,A -85,B 0,C 180,E1 -25332.757,E2 -25332.757} C_VEL
LIN {X 0,Y 131.001,Z 441.49,A -85,B 0,C 180,E1 -25334.319,E2 -25334.319} C_VEL
LIN {X 0,Y 129.822,Z 437.966,A -85,B 0,C 180,E1 -25335.112,E2 -25335.112} C_VEL
LIN {X 0,Y 129.217,Z 434.4,A -85,B 0,C 180,E1 -25341.966,E2 -25341.966} C_VEL
LIN {X 0,Y 129.004,Z 434.417,A -85,B 0,C 180,E1 -25346.989,E2 -25346.989} C_VEL
LIN {X 0,Y 129.054,Z 434.402,A -85,B 0,C 180,E1 -25350.651,E2 -25350.651} C_VEL
LIN {X 0,Y 129.051,Z 434.402,A -85,B 0,C 180,E1 -25356.796,E2 -25356.796} C_VEL
LIN {X 0,Y 128.538,Z 434.483,A -85,B 0,C 180,E1 -25359.402,E2 -25359.402} C_VEL
LIN {X 0,Y 127.103,Z 434.668,A -85,B 0,C 180,E1 -25361.981,E2 -25361.981} C_VEL
LIN {X 0,Y 122.752,Z 435.191,A -85,B 0,C 180,E1 -25369.095,E2 -25369.095} C_VEL
LIN {X 0,Y 122.409,Z 435.228,A -85,B 0,C 180,E1 -25370.973,E2 -25370.973} C_VEL
LIN {X 0,Y 123.045,Z 435.155,A -85,B 0,C 180,E1 -25380,E2 -25380} C_VEL
LIN {X 0,Y 122.419,Z 435.225,A -85,B 0,C 180,E1 -25387.166,E2 -25387.166} C_VEL
LIN {X 0,Y 122.366,Z 435.232,A -85,B 0,C 180,E1 -25392.473,E2 -25392.473} C_VEL
LIN {X 0,Y 122.048,Z 435.25,A -85,B 0,C 180,E1 -25400.212,E2 -25400.212} C_VEL
LIN {X 0,Y 121.986,Z 435.283,A -85,B 0,C 180,E1 -25403.784,E2 -25403.784} C_VEL
LIN {X 0,Y 121.943,Z 435.289,A -85,B 0,C 180,E1 -25410.173,E2 -25410.173} C_VEL
LIN {X 0,Y 121.898,Z 435.263,A -85,B 0,C 180,E1 -25416.179,E2 -25416.179} C_VEL
LIN {X 0,Y 121.866,Z 435.301,A -85,B 0,C 180,E1 -25421.433,E2 -25421.433} C_VEL
LIN {X 0,Y 121.885,Z 435.285,A -85,B 0,C 180,E1 -25428.555,E2 -25428.555} C_VEL
LIN {X 0,Y 121.947,Z 435.288,A -85,B 0,C 180,E1 -25434.807,E2 -25434.807} C_VEL
LIN {X 0,Y 121.944,Z 435.291,A -85,B 0,C 180,E1 -25439.825,E2 -25439.825} C_VEL
LIN {X 0,Y 121.985,Z 435.287,A -85,B 0,C 180,E1 -25446.214,E2 -25446.214} C_VEL
LIN {X 0,Y 122.051,Z 435.278,A -85,B 0,C 180,E1 -25449.787,E2 -25449.787} C_VEL
LIN {X 0,Y 122.266,Z 435.256,A -85,B 0,C 180,E1 -25456.706,E2 -25456.706} C_VEL
LIN {X 0,Y 122.458,Z 435.228,A -85,B 0,C 180,E1 -25460.085,E2 -25460.085} C_VEL
LIN {X 0,Y 122.605,Z 435.194,A -85,B 0,C 180,E1 -25466.61,E2 -25466.61} C_VEL
LIN {X 0,Y 123.744,Z 438.098,A -85,B 0,C 180,E1 -25467.405,E2 -25467.405} C_VEL
LIN {X 0,Y 125.033,Z 440.378,A -85,B 0,C 180,E1 -25468.138,E2 -25468.138} C_VEL
LIN {X 0,Y 127.789,Z 446.934,A -85,B 0,C 180,E1 -25469.999,E2 -25469.999} C_VEL
LIN {X 0,Y 130.458,Z 454.897,A -85,B 0,C 180,E1 -25472.237,E2 -25472.237} C_VEL
LIN {X 0,Y 132.103,Z 465.15,A -85,B 0,C 180,E1 -25474.983,E2 -25474.983} C_VEL
LIN {X 0,Y 133.209,Z 476.261,A -85,B 0,C 180,E1 -25478.341,E2 -25478.341} C_VEL
LIN {X 0,Y 133.502,Z 481.934,A -85,B 0,C 180,E1 -25480.233,E2 -25480.233} C_VEL
LIN {X 0,Y 130.186,Z 492.364,A -85,B 0,C 180,E1 -25483.659,E2 -25483.659} C_VEL
LIN {X 0,Y 126.893,Z 502.032,A -85,B 0,C 180,E1 -25487.734,E2 -25487.734} C_VEL
LIN {X 0,Y 123.998,Z 510.716,A -85,B 0,C 180,E1 -25492.492,E2 -25492.492} C_VEL
LIN {X 0,Y 121.73,Z 517.781,A -85,B 0,C 180,E1 -25497.507,E2 -25497.507} C_VEL
LIN {X 0,Y 120.067,Z 523.951,A -85,B 0,C 180,E1 -25503.215,E2 -25503.215} C_VEL
LIN {X 0,Y 119.193,Z 527.804,A -85,B 0,C 180,E1 -25507.916,E2 -25507.916} C_VEL
LIN {X 0,Y 118.852,Z 530.775,A -85,B 0,C 180,E1 -25512.662,E2 -25512.662} C_VEL
LIN {X 0,Y 119.54,Z 533.756,A -85,B 0,C 180,E1 -25519.842,E2 -25519.842} C_VEL
LIN {X 0,Y 120.802,Z 534.762,A -85,B 0,C 180,E1 -25524.534,E2 -25524.534} C_VEL
LIN {X 0,Y 122.785,Z 534.999,A -85,B 0,C 180,E1 -25529.154,E2 -25529.154} C_VEL
LIN {X 0,Y 125.436,Z 534.498,A -85,B 0,C 180,E1 -25533.692,E2 -25533.692} C_VEL
LIN {X 0,Y 128.809,Z 533.233,A -85,B 0,C 180,E1 -25538.051,E2 -25538.051} C_VEL
LIN {X 0,Y 134.518,Z 530.135,A -85,B 0,C 180,E1 -25543.64,E2 -25543.64} C_VEL
LIN {X 0,Y 141.157,Z 525.683,A -85,B 0,C 180,E1 -25548.513,E2 -25548.513} C_VEL
LIN {X 0,Y 146.575,Z 521.414,A -85,B 0,C 180,E1 -25551.73,E2 -25551.73} C_VEL
LIN {X 0,Y 153.965,Z 514.706,A -85,B 0,C 180,E1 -25555.444,E2 -25555.444} C_VEL
LIN {X 0,Y 158.363,Z 510.057,A -85,B 0,C 180,E1 -25557.457,E2 -25557.457} C_VEL
LIN {X 0,Y 160.012,Z 506.436,A -85,B 0,C 180,E1 -25560,E2 -25560} C_VEL
LIN {X 0,Y 160.898,Z 503.374,A -85,B 0,C 180,E1 -25562.504,E2 -25562.504} C_VEL
LIN {X 0,Y 161.364,Z 499.692,A -85,B 0,C 180,E1 -25566.251,E2 -25566.251} C_VEL
LIN {X 0,Y 161.249,Z 497.052,A -85,B 0,C 180,E1 -25570.04,E2 -25570.04} C_VEL
LIN {X 0,Y 161.072,Z 494.821,A -85,B 0,C 180,E1 -25575.177,E2 -25575.177} C_VEL
LIN {X 0,Y 160.391,Z 494.867,A -85,B 0,C 180,E1 -25580.521,E2 -25580.521} C_VEL
LIN {X 0,Y 160.443,Z 496.17,A -85,B 0,C 180,E1 -25585.979,E2 -25585.979} C_VEL
LIN {X 0,Y 160.359,Z 499.809,A -85,B 0,C 180,E1 -25591.73,E2 -25591.73} C_VEL
LIN {X 0,Y 160.231,Z 502.589,A -85,B 0,C 180,E1 -25594.765,E2 -25594.765} C_VEL
LIN {X 0,Y 159.874,Z 506.134,A -85,B 0,C 180,E1 -25597.984,E2 -25597.984} C_VEL
LIN {X 0,Y 159.259,Z 508.79,A -85,B 0,C 180,E1 -25599.989,E2 -25599.989} C_VEL
LIN {X 0,Y 156.59,Z 513.88,A -85,B 0,C 180,E1 -25602.824,E2 -25602.824} C_VEL
LIN {X 0,Y 153.302,Z 518.971,A -85,B 0,C 180,E1 -25605.645,E2 -25605.645} C_VEL
LIN {X 0,Y 151.455,Z 521.22,A -85,B 0,C 180,E1 -25606.81,E2 -25606.81} C_VEL
LIN {X 0,Y 143.886,Z 528.19,A -85,B 0,C 180,E1 -25610.584,E2 -25610.584} C_VEL
LIN {X 0,Y 138.107,Z 532.942,A -85,B 0,C 180,E1 -25614.184,E2 -25614.184} C_VEL
LIN {X 0,Y 133.085,Z 536.72,A -85,B 0,C 180,E1 -25618.126,E2 -25618.126} C_VEL
LIN {X 0,Y 127.419,Z 540.336,A -85,B 0,C 180,E1 -25623.818,E2 -25623.818} C_VEL
LIN {X 0,Y 123.061,Z 542.445,A -85,B 0,C 180,E1 -25629.962,E2 -25629.962} C_VEL
LIN {X 0,Y 120.534,Z 543.078,A -85,B 0,C 180,E1 -25636.514,E2 -25636.514} C_VEL
LIN {X 0,Y 119.483,Z 542.282,A -85,B 0,C 180,E1 -25643.245,E2 -25643.245} C_VEL
LIN {X 0,Y 119.533,Z 540.692,A -85,B 0,C 180,E1 -25648.24,E2 -25648.24} C_VEL
LIN {X 0,Y 119.554,Z 538.861,A -85,B 0,C 180,E1 -25652.066,E2 -25652.066} C_VEL
LIN {X 0,Y 119.628,Z 535.766,A -85,B 0,C 180,E1 -25656.749,E2 -25656.749} C_VEL
LIN {X 0,Y 120.261,Z 531.338,A -85,B 0,C 180,E1 -25661.804,E2 -25661.804} C_VEL
LIN {X 0,Y 121.884,Z 524.564,A -85,B 0,C 180,E1 -25667.622,E2 -25667.622} C_VEL
LIN {X 0,Y 124.226,Z 517.212,A -85,B 0,C 180,E1 -25672.451,E2 -25672.451} C_VEL
LIN {X 0,Y 127.198,Z 508.15,A -85,B 0,C 180,E1 -25677.062,E2 -25677.062} C_VEL
LIN {X 0,Y 129.961,Z 500.122,A -85,B 0,C 180,E1 -25680.261,E2 -25680.261} C_VEL
LIN {X 0,Y 130.579,Z 493.773,A -85,B 0,C 180,E1 -25682.564,E2 -25682.564} C_VEL
LIN {X 0,Y 130.783,Z 482.18,A -85,B 0,C 180,E1 -25686.286,E2 -25686.286} C_VEL
LIN {X 0,Y 130.44,Z 470.038,A -85,B 0,C 180,E1 -25689.528,E2 -25689.528} C_VEL
LIN {X 0,Y 129.436,Z 458.303,A -85,B 0,C 180,E1 -25692.202,E2 -25692.202} C_VEL
LIN {X 0,Y 128.282,Z 453.055,A -85,B 0,C 180,E1 -25693.401,E2 -25693.401} C_VEL
LIN {X 0,Y 124.06,Z 441.765,A -85,B 0,C 180,E1 -25696.195,E2 -25696.195} C_VEL
LIN {X 0,Y 122.72,Z 438.603,A -85,B 0,C 180,E1 -25696.983,E2 -25696.983} C_VEL
LIN {X 0,Y 122.537,Z 437.665,A -85,B 0,C 180,E1 -25697.295,E2 -25697.295} C_VEL
LIN {X 0,Y 122.129,Z 435.266,A -85,B 0,C 180,E1 -25702.406,E2 -25702.406} C_VEL
LIN {X 0,Y 121.945,Z 435.294,A -85,B 0,C 180,E1 -25709.826,E2 -25709.826} C_VEL
LIN {X 0,Y 121.986,Z 435.287,A -85,B 0,C 180,E1 -25716.216,E2 -25716.216} C_VEL
LIN {X 0,Y 122.052,Z 435.28,A -85,B 0,C 180,E1 -25719.788,E2 -25719.788} C_VEL
LIN {X 0,Y 122.267,Z 435.252,A -85,B 0,C 180,E1 -25726.707,E2 -25726.707} C_VEL
LIN {X 0,Y 122.409,Z 435.228,A -85,B 0,C 180,E1 -25730.973,E2 -25730.973} C_VEL
LIN {X 0,Y 121.703,Z 435.322,A -85,B 0,C 180,E1 -25733.73,E2 -25733.73} C_VEL
LIN {X 0,Y 120.144,Z 435.514,A -85,B 0,C 180,E1 -25736.455,E2 -25736.455} C_VEL
LIN {X 0,Y 115.709,Z 436.061,A -85,B 0,C 180,E1 -25744.003,E2 -25744.003} C_VEL
LIN {X 0,Y 115.387,Z 436.099,A -85,B 0,C 180,E1 -25746.001,E2 -25746.001} C_VEL
LIN {X 0,Y 115.388,Z 436.108,A -85,B 0,C 180,E1 -25750.528,E2 -25750.528} C_VEL
LIN {X 0,Y 115.148,Z 436.121,A -85,B 0,C 180,E1 -25754.131,E2 -25754.131} C_VEL
LIN {X 0,Y 114.982,Z 436.139,A -85,B 0,C 180,E1 -25761.514,E2 -25761.514} C_VEL
LIN {X 0,Y 114.876,Z 436.174,A -85,B 0,C 180,E1 -25765.357,E2 -25765.357} C_VEL
LIN {X 0,Y 114.869,Z 436.166,A -85,B 0,C 180,E1 -25771.066,E2 -25771.066} C_VEL
LIN {X 0,Y 114.786,Z 436.156,A -85,B 0,C 180,E1 -25777.754,E2 -25777.754} C_VEL
LIN {X 0,Y 114.782,Z 436.185,A -85,B 0,C 180,E1 -25782.712,E2 -25782.712} C_VEL
LIN {X 0,Y 114.803,Z 436.173,A -85,B 0,C 180,E1 -25787.669,E2 -25787.669} C_VEL
LIN {X 0,Y 114.813,Z 436.162,A -85,B 0,C 180,E1 -25792.727,E2 -25792.727} C_VEL
LIN {X 0,Y 114.871,Z 436.174,A -85,B 0,C 180,E1 -25798.931,E2 -25798.931} C_VEL
LIN {X 0,Y 114.949,Z 436.165,A -85,B 0,C 180,E1 -25806.506,E2 -25806.506} C_VEL
LIN {X 0,Y 115.02,Z 436.147,A -85,B 0,C 180,E1 -25812.21,E2 -25812.21} C_VEL
LIN {X 0,Y 115.288,Z 436.124,A -85,B 0,C 180,E1 -25817.256,E2 -25817.256} C_VEL
LIN {X 0,Y 115.398,Z 436.108,A -85,B 0,C 180,E1 -25823.002,E2 -25823.002} C_VEL
LIN {X 0,Y 115.436,Z 436.091,A -85,B 0,C 180,E1 -25824.43,E2 -25824.43} C_VEL
LIN {X 0,Y 116.477,Z 438.95,A -85,B 0,C 180,E1 -25825.24,E2 -25825.24} C_VEL
LIN {X 0,Y 117.809,Z 441.182,A -85,B 0,C 180,E1 -25826.044,E2 -25826.044} C_VEL
LIN {X 0,Y 120.986,Z 447.472,A -85,B 0,C 180,E1 -25828.168,E2 -25828.168} C_VEL
LIN {X 0,Y 124.248,Z 457.593,A -85,B 0,C 180,E1 -25831.268,E2 -25831.268} C_VEL
LIN {X 0,Y 125.885,Z 469.509,A -85,B 0,C 180,E1 -25834.803,E2 -25834.803} C_VEL
LIN {X 0,Y 126.658,Z 480.204,A -85,B 0,C 180,E1 -25838.374,E2 -25838.374} C_VEL
LIN {X 0,Y 126.738,Z 482.447,A -85,B 0,C 180,E1 -25839.172,E2 -25839.172} C_VEL
LIN {X 0,Y 123.36,Z 492.766,A -85,B 0,C 180,E1 -25842.753,E2 -25842.753} C_VEL
LIN {X 0,Y 119.925,Z 502.394,A -85,B 0,C 180,E1 -25847.037,E2 -25847.037} C_VEL
LIN {X 0,Y 116.919,Z 511.04,A -85,B 0,C 180,E1 -25852.065,E2 -25852.065} C_VEL
LIN {X 0,Y 114.585,Z 518.095,A -85,B 0,C 180,E1 -25857.386,E2 -25857.386} C_VEL
LIN {X 0,Y 113.242,Z 522.89,A -85,B 0,C 180,E1 -25861.962,E2 -25861.962} C_VEL
LIN {X 0,Y 112.221,Z 527.182,A -85,B 0,C 180,E1 -25867.136,E2 -25867.136} C_VEL
LIN {X 0,Y 111.751,Z 531.214,A -85,B 0,C 180,E1 -25873.769,E2 -25873.769} C_VEL
LIN {X 0,Y 112.216,Z 533.294,A -85,B 0,C 180,E1 -25878.722,E2 -25878.722} C_VEL
LIN {X 0,Y 113.351,Z 534.672,A -85,B 0,C 180,E1 -25883.707,E2 -25883.707} C_VEL
LIN {X 0,Y 115.243,Z 535.277,A -85,B 0,C 180,E1 -25888.622,E2 -25888.622} C_VEL
LIN {X 0,Y 119.382,Z 534.816,A -85,B 0,C 180,E1 -25895.664,E2 -25895.664} C_VEL
LIN {X 0,Y 122.861,Z 533.656,A -85,B 0,C 180,E1 -25899.927,E2 -25899.927} C_VEL
LIN {X 0,Y 126.972,Z 531.759,A -85,B 0,C 180,E1 -25903.934,E2 -25903.934} C_VEL
LIN {X 0,Y 133.772,Z 527.892,A -85,B 0,C 180,E1 -25909.09,E2 -25909.09} C_VEL
LIN {X 0,Y 139.425,Z 523.992,A -85,B 0,C 180,E1 -25912.533,E2 -25912.533} C_VEL
LIN {X 0,Y 145.51,Z 519.157,A -85,B 0,C 180,E1 -25915.696,E2 -25915.696} C_VEL
LIN {X 0,Y 152.236,Z 513.085,A -85,B 0,C 180,E1 -25918.678,E2 -25918.678} C_VEL
LIN {X 0,Y 153.224,Z 511.931,A -85,B 0,C 180,E1 -25919.343,E2 -25919.343} C_VEL
LIN {X 0,Y 154.665,Z 509.203,A -85,B 0,C 180,E1 -25921.505,E2 -25921.505} C_VEL
LIN {X 0,Y 155.507,Z 506.662,A -85,B 0,C 180,E1 -25923.887,E2 -25923.887} C_VEL
LIN {X 0,Y 156.02,Z 504.415,A -85,B 0,C 180,E1 -25926.466,E2 -25926.466} C_VEL
LIN {X 0,Y 156.183,Z 501.921,A -85,B 0,C 180,E1 -25930.37,E2 -25930.37} C_VEL
LIN {X 0,Y 156.114,Z 499.971,A -85,B 0,C 180,E1 -25935.671,E2 -25935.671} C_VEL
LIN {X 0,Y 155.542,Z 500.207,A -85,B 0,C 180,E1 -25941.191,E2 -25941.191} C_VEL
LIN {X 0,Y 155.524,Z 501.168,A -85,B 0,C 180,E1 -25945.343,E2 -25945.343} C_VEL
LIN {X 0,Y 155.202,Z 504.139,A -85,B 0,C 180,E1 -25950.644,E2 -25950.644} C_VEL
LIN {X 0,Y 154.948,Z 506.541,A -85,B 0,C 180,E1 -25953.696,E2 -25953.696} C_VEL
LIN {X 0,Y 154.524,Z 509.003,A -85,B 0,C 180,E1 -25956.247,E2 -25956.247} C_VEL
LIN {X 0,Y 154.106,Z 510.768,A -85,B 0,C 180,E1 -25957.894,E2 -25957.894} C_VEL
LIN {X 0,Y 153.622,Z 512.122,A -85,B 0,C 180,E1 -25958.949,E2 -25958.949} C_VEL
LIN {X 0,Y 149.903,Z 517.88,A -85,B 0,C 180,E1 -25962.405,E2 -25962.405} C_VEL
LIN {X 0,Y 147.387,Z 521.094,A -85,B 0,C 180,E1 -25964.338,E2 -25964.338} C_VEL
LIN {X 0,Y 142.94,Z 525.214,A -85,B 0,C 180,E1 -25966.503,E2 -25966.503} C_VEL
LIN {X 0,Y 136.407,Z 530.497,A -85,B 0,C 180,E1 -25969.909,E2 -25969.909} C_VEL
LIN {X 0,Y 129.492,Z 535.451,A -85,B 0,C 180,E1 -25974.499,E2 -25974.499} C_VEL
LIN {X 0,Y 123.918,Z 538.887,A -85,B 0,C 180,E1 -25979.309,E2 -25979.309} C_VEL
LIN {X 0,Y 118.535,Z 541.525,A -85,B 0,C 180,E1 -25985.48,E2 -25985.48} C_VEL
LIN {X 0,Y 114.802,Z 542.7,A -85,B 0,C 180,E1 -25992.178,E2 -25992.178} C_VEL
LIN {X 0,Y 112.834,Z 542.468,A -85,B 0,C 180,E1 -25999.232,E2 -25999.232} C_VEL
LIN {X 0,Y 112.398,Z 540.705,A -85,B 0,C 180,E1 -26006.416,E2 -26006.416} C_VEL
LIN {X 0,Y 112.577,Z 539.237,A -85,B 0,C 180,E1 -26010.001,E2 -26010.001} C_VEL
LIN {X 0,Y 112.496,Z 536.128,A -85,B 0,C 180,E1 -26015.378,E2 -26015.378} C_VEL
LIN {X 0,Y 112.996,Z 531.925,A -85,B 0,C 180,E1 -26020.755,E2 -26020.755} C_VEL
LIN {X 0,Y 114.476,Z 525.505,A -85,B 0,C 180,E1 -26026.956,E2 -26026.956} C_VEL
LIN {X 0,Y 116.728,Z 518.443,A -85,B 0,C 180,E1 -26032.106,E2 -26032.106} C_VEL
LIN {X 0,Y 119.72,Z 509.648,A -85,B 0,C 180,E1 -26037.063,E2 -26037.063} C_VEL
LIN {X 0,Y 123.033,Z 500.507,A -85,B 0,C 180,E1 -26041.035,E2 -26041.035} C_VEL
LIN {X 0,Y 123.626,Z 496.294,A -85,B 0,C 180,E1 -26042.687,E2 -26042.687} C_VEL
LIN {X 0,Y 124.043,Z 486.449,A -85,B 0,C 180,E1 -26046.194,E2 -26046.194} C_VEL
LIN {X 0,Y 124.02,Z 474.293,A -85,B 0,C 180,E1 -26049.834,E2 -26049.834} C_VEL
LIN {X 0,Y 123.398,Z 462.811,A -85,B 0,C 180,E1 -26052.777,E2 -26052.777} C_VEL
LIN {X 0,Y 122.531,Z 457.054,A -85,B 0,C 180,E1 -26054.193,E2 -26054.193} C_VEL
LIN {X 0,Y 119.407,Z 447.917,A -85,B 0,C 180,E1 -26056.718,E2 -26056.718} C_VEL
LIN {X 0,Y 116.464,Z 440.883,A -85,B 0,C 180,E1 -26058.698,E2 -26058.698} C_VEL
LIN {X 0,Y 115.287,Z 437.403,A -85,B 0,C 180,E1 -26059.63,E2 -26059.63} C_VEL
LIN {X 0,Y 115.077,Z 436.142,A -85,B 0,C 180,E1 -26062.557,E2 -26062.557} C_VEL
LIN {X 0,Y 114.876,Z 436.167,A -85,B 0,C 180,E1 -26070.696,E2 -26070.696} C_VEL
LIN {X 0,Y 114.95,Z 436.164,A -85,B 0,C 180,E1 -26076.508,E2 -26076.508} C_VEL
LIN {X 0,Y 115.021,Z 436.152,A -85,B 0,C 180,E1 -26082.211,E2 -26082.211} C_VEL
LIN {X 0,Y 115.287,Z 436.118,A -85,B 0,C 180,E1 -26087.262,E2 -26087.262} C_VEL
LIN {X 0,Y 115.391,Z 436.11,A -85,B 0,C 180,E1 -26093.003,E2 -26093.003} C_VEL
LIN {X 0,Y 115.997,Z 436.033,A -85,B 0,C 180,E1 -26100,E2 -26100} C_VEL
LIN {X 0,Y 115.387,Z 436.099,A -85,B 0,C 180,E1 -26106.001,E2 -26106.001} C_VEL
LIN {X 0,Y 114.636,Z 436.203,A -85,B 0,C 180,E1 -26108.907,E2 -26108.907} C_VEL
LIN {X 0,Y 112.927,Z 436.411,A -85,B 0,C 180,E1 -26111.773,E2 -26111.773} C_VEL
LIN {X 0,Y 108.136,Z 436.975,A -85,B 0,C 180,E1 -26119.763,E2 -26119.763} C_VEL
LIN {X 0,Y 107.859,Z 437.021,A -85,B 0,C 180,E1 -26121.898,E2 -26121.898} C_VEL
LIN {X 0,Y 107.764,Z 437.061,A -85,B 0,C 180,E1 -26127.162,E2 -26127.162} C_VEL
LIN {X 0,Y 107.793,Z 437.039,A -85,B 0,C 180,E1 -26132.048,E2 -26132.048} C_VEL
LIN {X 0,Y 107.693,Z 437.044,A -85,B 0,C 180,E1 -26138.451,E2 -26138.451} C_VEL
LIN {X 0,Y 107.681,Z 437.068,A -85,B 0,C 180,E1 -26145.884,E2 -26145.884} C_VEL
LIN {X 0,Y 107.707,Z 437.04,A -85,B 0,C 180,E1 -26151.537,E2 -26151.537} C_VEL
LIN {X 0,Y 107.809,Z 437.055,A -85,B 0,C 180,E1 -26158.565,E2 -26158.565} C_VEL
LIN {X 0,Y 107.913,Z 437.044,A -85,B 0,C 180,E1 -26166.997,E2 -26166.997} C_VEL
LIN {X 0,Y 108.041,Z 437.03,A -85,B 0,C 180,E1 -26174.917,E2 -26174.917} C_VEL
LIN {X 0,Y 108.306,Z 436.993,A -85,B 0,C 180,E1 -26180.663,E2 -26180.663} C_VEL
LIN {X 0,Y 108.314,Z 436.995,A -85,B 0,C 180,E1 -26181.839,E2 -26181.839} C_VEL
LIN {X 0,Y 109.373,Z 439.884,A -85,B 0,C 180,E1 -26182.847,E2 -26182.847} C_VEL
LIN {X 0,Y 110.504,Z 441.711,A -85,B 0,C 180,E1 -26183.609,E2 -26183.609} C_VEL
LIN {X 0,Y 115.06,Z 450.657,A -85,B 0,C 180,E1 -26187.022,E2 -26187.022} C_VEL
LIN {X 0,Y 117.912,Z 459.51,A -85,B 0,C 180,E1 -26189.999,E2 -26189.999} C_VEL
LIN {X 0,Y 119.362,Z 471.279,A -85,B 0,C 180,E1 -26193.797,E2 -26193.797} C_VEL
LIN {X 0,Y 119.948,Z 481.761,A -85,B 0,C 180,E1 -26197.574,E2 -26197.574} C_VEL
LIN {X 0,Y 119.726,Z 484.085,A -85,B 0,C 180,E1 -26198.437,E2 -26198.437} C_VEL
LIN {X 0,Y 116.141,Z 494.182,A -85,B 0,C 180,E1 -26202.191,E2 -26202.191} C_VEL
LIN {X 0,Y 113.002,Z 502.699,A -85,B 0,C 180,E1 -26206.251,E2 -26206.251} C_VEL
LIN {X 0,Y 110.363,Z 509.938,A -85,B 0,C 180,E1 -26210.602,E2 -26210.602} C_VEL
LIN {X 0,Y 107.942,Z 516.891,A -85,B 0,C 180,E1 -26215.874,E2 -26215.874} C_VEL
LIN {X 0,Y 106.102,Z 523.085,A -85,B 0,C 180,E1 -26221.997,E2 -26221.997} C_VEL
LIN {X 0,Y 105.145,Z 527.026,A -85,B 0,C 180,E1 -26226.98,E2 -26226.98} C_VEL
LIN {X 0,Y 104.686,Z 531.519,A -85,B 0,C 180,E1 -26234.817,E2 -26234.817} C_VEL
LIN {X 0,Y 104.982,Z 532.849,A -85,B 0,C 180,E1 -26237.976,E2 -26237.976} C_VEL
LIN {X 0,Y 106.083,Z 534.523,A -85,B 0,C 180,E1 -26243.398,E2 -26243.398} C_VEL
LIN {X 0,Y 107.953,Z 535.442,A -85,B 0,C 180,E1 -26248.613,E2 -26248.613} C_VEL
LIN {X 0,Y 110.545,Z 535.598,A -85,B 0,C 180,E1 -26253.575,E2 -26253.575} C_VEL
LIN {X 0,Y 113.821,Z 535.059,A -85,B 0,C 180,E1 -26258.255,E2 -26258.255} C_VEL
LIN {X 0,Y 117.778,Z 533.847,A -85,B 0,C 180,E1 -26262.691,E2 -26262.691} C_VEL
LIN {X 0,Y 124.956,Z 530.589,A -85,B 0,C 180,E1 -26268.77,E2 -26268.77} C_VEL
LIN {X 0,Y 133.196,Z 525.762,A -85,B 0,C 180,E1 -26273.943,E2 -26273.943} C_VEL
LIN {X 0,Y 140.669,Z 520.416,A -85,B 0,C 180,E1 -26277.711,E2 -26277.711} C_VEL
LIN {X 0,Y 147.595,Z 514.607,A -85,B 0,C 180,E1 -26280.698,E2 -26280.698} C_VEL
LIN {X 0,Y 149.075,Z 512.315,A -85,B 0,C 180,E1 -26282.702,E2 -26282.702} C_VEL
LIN {X 0,Y 150.109,Z 509.918,A -85,B 0,C 180,E1 -26285.373,E2 -26285.373} C_VEL
LIN {X 0,Y 150.653,Z 507.968,A -85,B 0,C 180,E1 -26288.045,E2 -26288.045} C_VEL
LIN {X 0,Y 150.893,Z 506.54,A -85,B 0,C 180,E1 -26290.737,E2 -26290.737} C_VEL
LIN {X 0,Y 150.908,Z 505.529,A -85,B 0,C 180,E1 -26293.466,E2 -26293.466} C_VEL
LIN {X 0,Y 150.9,Z 504.894,A -85,B 0,C 180,E1 -26296.227,E2 -26296.227} C_VEL
LIN {X 0,Y 150.382,Z 505.317,A -85,B 0,C 180,E1 -26301.955,E2 -26301.955} C_VEL
LIN {X 0,Y 150.379,Z 505.952,A -85,B 0,C 180,E1 -26304.874,E2 -26304.874} C_VEL
LIN {X 0,Y 150.026,Z 507.403,A -85,B 0,C 180,E1 -26307.934,E2 -26307.934} C_VEL
LIN {X 0,Y 149.597,Z 510.057,A -85,B 0,C 180,E1 -26312.263,E2 -26312.263} C_VEL
LIN {X 0,Y 149.178,Z 511.855,A -85,B 0,C 180,E1 -26314.426,E2 -26314.426} C_VEL
LIN {X 0,Y 148.582,Z 513.792,A -85,B 0,C 180,E1 -26316.478,E2 -26316.478} C_VEL
LIN {X 0,Y 147.865,Z 515.359,A -85,B 0,C 180,E1 -26317.894,E2 -26317.894} C_VEL
LIN {X 0,Y 144.254,Z 520.12,A -85,B 0,C 180,E1 -26320.963,E2 -26320.963} C_VEL
LIN {X 0,Y 141.5,Z 523.138,A -85,B 0,C 180,E1 -26322.897,E2 -26322.897} C_VEL
LIN {X 0,Y 133.299,Z 529.521,A -85,B 0,C 180,E1 -26326.734,E2 -26326.734} C_VEL
LIN {X 0,Y 124.921,Z 535.109,A -85,B 0,C 180,E1 -26331.769,E2 -26331.769} C_VEL
LIN {X 0,Y 121.247,Z 537.285,A -85,B 0,C 180,E1 -26334.576,E2 -26334.576} C_VEL
LIN {X 0,Y 114.798,Z 540.424,A -85,B 0,C 180,E1 -26340.677,E2 -26340.677} C_VEL
LIN {X 0,Y 109.794,Z 542.131,A -85,B 0,C 180,E1 -26347.416,E2 -26347.416} C_VEL
LIN {X 0,Y 106.749,Z 542.416,A -85,B 0,C 180,E1 -26354.733,E2 -26354.733} C_VEL
LIN {X 0,Y 105.402,Z 541.226,A -85,B 0,C 180,E1 -26362.338,E2 -26362.338} C_VEL
LIN {X 0,Y 105.446,Z 539.088,A -85,B 0,C 180,E1 -26368.755,E2 -26368.755} C_VEL
LIN {X 0,Y 105.393,Z 536.485,A -85,B 0,C 180,E1 -26373.825,E2 -26373.825} C_VEL
LIN {X 0,Y 105.752,Z 532.493,A -85,B 0,C 180,E1 -26379.565,E2 -26379.565} C_VEL
LIN {X 0,Y 106.805,Z 527.295,A -85,B 0,C 180,E1 -26385.262,E2 -26385.262} C_VEL
LIN {X 0,Y 108.822,Z 520.762,A -85,B 0,C 180,E1 -26390.807,E2 -26390.807} C_VEL
LIN {X 0,Y 111.708,Z 512.646,A -85,B 0,C 180,E1 -26396.131,E2 -26396.131} C_VEL
LIN {X 0,Y 115.067,Z 503.502,A -85,B 0,C 180,E1 -26400.726,E2 -26400.726} C_VEL
LIN {X 0,Y 116.461,Z 499.637,A -85,B 0,C 180,E1 -26402.344,E2 -26402.344} C_VEL
LIN {X 0,Y 117.157,Z 491.085,A -85,B 0,C 180,E1 -26405.796,E2 -26405.796} C_VEL
LIN {X 0,Y 117.475,Z 479.822,A -85,B 0,C 180,E1 -26409.676,E2 -26409.676} C_VEL
LIN {X 0,Y 117.27,Z 468.16,A -85,B 0,C 180,E1 -26413.097,E2 -26413.097} C_VEL
LIN {X 0,Y 116.459,Z 459.874,A -85,B 0,C 180,E1 -26415.33,E2 -26415.33} C_VEL
LIN {X 0,Y 113.459,Z 450.706,A -85,B 0,C 180,E1 -26418.129,E2 -26418.129} C_VEL
LIN {X 0,Y 109.525,Z 441.013,A -85,B 0,C 180,E1 -26421.136,E2 -26421.136} C_VEL
LIN {X 0,Y 108.194,Z 437.814,A -85,B 0,C 180,E1 -26422.119,E2 -26422.119} C_VEL
LIN {X 0,Y 108.046,Z 437.08,A -85,B 0,C 180,E1 -26422.386,E2 -26422.386} C_VEL
LIN {X 0,Y 107.818,Z 437.058,A -85,B 0,C 180,E1 -26428.569,E2 -26428.569} C_VEL
LIN {X 0,Y 107.914,Z 437.041,A -85,B 0,C 180,E1 -26436.998,E2 -26436.998} C_VEL
LIN {X 0,Y 108.042,Z 437.027,A -85,B 0,C 180,E1 -26444.918,E2 -26444.918} C_VEL
LIN {X 0,Y 108.291,Z 436.987,A -85,B 0,C 180,E1 -26448.773,E2 -26448.773} C_VEL
LIN {X 0,Y 108.458,Z 436.963,A -85,B 0,C 180,E1 -26456.284,E2 -26456.284} C_VEL
LIN {X 0,Y 108.947,Z 436.911,A -85,B 0,C 180,E1 -26460,E2 -26460} C_VEL
LIN {X 0,Y 108.334,Z 436.986,A -85,B 0,C 180,E1 -26467.455,E2 -26467.455} C_VEL
LIN {X 0,Y 108.204,Z 436.992,A -85,B 0,C 180,E1 -26473.02,E2 -26473.02} C_VEL
LIN {X 0,Y 107.907,Z 436.999,A -85,B 0,C 180,E1 -26479.005,E2 -26479.005} C_VEL
LIN {X 0,Y 107.859,Z 437.021,A -85,B 0,C 180,E1 -26481.898,E2 -26481.898} C_VEL
LIN {X 0,Y 107.585,Z 437.077,A -85,B 0,C 180,E1 -26483.98,E2 -26483.98} C_VEL
LIN {X 0,Y 106.785,Z 437.182,A -85,B 0,C 180,E1 -26486.04,E2 -26486.04} C_VEL
LIN {X 0,Y 104.331,Z 437.482,A -85,B 0,C 180,E1 -26490.144,E2 -26490.144} C_VEL
LIN {X 0,Y 100.951,Z 437.881,A -85,B 0,C 180,E1 -26496.694,E2 -26496.694} C_VEL
LIN {X 0,Y 100.63,Z 437.928,A -85,B 0,C 180,E1 -26498.991,E2 -26498.991} C_VEL
LIN {X 0,Y 100.65,Z 437.945,A -85,B 0,C 180,E1 -26505.711,E2 -26505.711} C_VEL
LIN {X 0,Y 100.645,Z 437.918,A -85,B 0,C 180,E1 -26511.061,E2 -26511.061} C_VEL
LIN {X 0,Y 100.702,Z 437.942,A -85,B 0,C 180,E1 -26516.875,E2 -26516.875} C_VEL
LIN {X 0,Y 100.787,Z 437.921,A -85,B 0,C 180,E1 -26525.266,E2 -26525.266} C_VEL
LIN {X 0,Y 100.82,Z 437.923,A -85,B 0,C 180,E1 -26529.6,E2 -26529.6} C_VEL
LIN {X 0,Y 101.193,Z 437.874,A -85,B 0,C 180,E1 -26537.973,E2 -26537.973} C_VEL
LIN {X 0,Y 101.265,Z 437.864,A -85,B 0,C 180,E1 -26538.996,E2 -26538.996} C_VEL
LIN {X 0,Y 102.234,Z 440.653,A -85,B 0,C 180,E1 -26540.04,E2 -26540.04} C_VEL
LIN {X 0,Y 103.625,Z 442.978,A -85,B 0,C 180,E1 -26541.098,E2 -26541.098} C_VEL
LIN {X 0,Y 108.403,Z 452.172,A -85,B 0,C 180,E1 -26545.112,E2 -26545.112} C_VEL
LIN {X 0,Y 111.005,Z 459.776,A -85,B 0,C 180,E1 -26548.003,E2 -26548.003} C_VEL
LIN {X 0,Y 112.01,Z 464.359,A -85,B 0,C 180,E1 -26549.639,E2 -26549.639} C_VEL
LIN {X 0,Y 112.895,Z 474.113,A -85,B 0,C 180,E1 -26553.076,E2 -26553.076} C_VEL
LIN {X 0,Y 113.27,Z 483.788,A -85,B 0,C 180,E1 -26556.906,E2 -26556.906} C_VEL
LIN {X 0,Y 109.336,Z 494.593,A -85,B 0,C 180,E1 -26561.117,E2 -26561.117} C_VEL
LIN {X 0,Y 106.081,Z 502.995,A -85,B 0,C 180,E1 -26565.366,E2 -26565.366} C_VEL
LIN {X 0,Y 102.779,Z 511.628,A -85,B 0,C 180,E1 -26571.037,E2 -26571.037} C_VEL
LIN {X 0,Y 100.256,Z 518.811,A -85,B 0,C 180,E1 -26577.234,E2 -26577.234} C_VEL
LIN {X 0,Y 98.696,Z 524.06,A -85,B 0,C 180,E1 -26583.091,E2 -26583.091} C_VEL
LIN {X 0,Y 97.635,Z 529.016,A -85,B 0,C 180,E1 -26590.377,E2 -26590.377} C_VEL
LIN {X 0,Y 97.662,Z 531.82,A -85,B 0,C 180,E1 -26596.021,E2 -26596.021} C_VEL
LIN {X 0,Y 98.487,Z 533.908,A -85,B 0,C 180,E1 -26601.714,E2 -26601.714} C_VEL
LIN {X 0,Y 100.154,Z 535.281,A -85,B 0,C 180,E1 -26607.355,E2 -26607.355} C_VEL
LIN {X 0,Y 102.695,Z 535.885,A -85,B 0,C 180,E1 -26612.827,E2 -26612.827} C_VEL
LIN {X 0,Y 106.051,Z 535.756,A -85,B 0,C 180,E1 -26618.086,E2 -26618.086} C_VEL
LIN {X 0,Y 110.223,Z 534.888,A -85,B 0,C 180,E1 -26623.017,E2 -26623.017} C_VEL
LIN {X 0,Y 115.14,Z 533.245,A -85,B 0,C 180,E1 -26627.577,E2 -26627.577} C_VEL
LIN {X 0,Y 123.537,Z 529.383,A -85,B 0,C 180,E1 -26633.467,E2 -26633.467} C_VEL
LIN {X 0,Y 131.883,Z 524.491,A -85,B 0,C 180,E1 -26637.964,E2 -26637.964} C_VEL
LIN {X 0,Y 140.622,Z 518.211,A -85,B 0,C 180,E1 -26641.749,E2 -26641.749} C_VEL
LIN {X 0,Y 142.652,Z 516.448,A -85,B 0,C 180,E1 -26642.824,E2 -26642.824} C_VEL
LIN {X 0,Y 144.167,Z 514.05,A -85,B 0,C 180,E1 -26645.595,E2 -26645.595} C_VEL
LIN {X 0,Y 144.954,Z 512.202,A -85,B 0,C 180,E1 -26648.364,E2 -26648.364} C_VEL
LIN {X 0,Y 145.353,Z 510.884,A -85,B 0,C 180,E1 -26651.152,E2 -26651.152} C_VEL
LIN {X 0,Y 145.454,Z 509.805,A -85,B 0,C 180,E1 -26654.91,E2 -26654.91} C_VEL
LIN {X 0,Y 145.447,Z 509.561,A -85,B 0,C 180,E1 -26656.853,E2 -26656.853} C_VEL
LIN {X 0,Y 145.159,Z 509.69,A -85,B 0,C 180,E1 -26659.811,E2 -26659.811} C_VEL
LIN {X 0,Y 144.983,Z 510.184,A -85,B 0,C 180,E1 -26662.928,E2 -26662.928} C_VEL
LIN {X 0,Y 144.777,Z 511.059,A -85,B 0,C 180,E1 -26665.906,E2 -26665.906} C_VEL
LIN {X 0,Y 144.093,Z 513.575,A -85,B 0,C 180,E1 -26670.806,E2 -26670.806} C_VEL
LIN {X 0,Y 143.206,Z 516.197,A -85,B 0,C 180,E1 -26674.358,E2 -26674.358} C_VEL
LIN {X 0,Y 142.35,Z 517.974,A -85,B 0,C 180,E1 -26676.332,E2 -26676.332} C_VEL
LIN {X 0,Y 139.606,Z 521.188,A -85,B 0,C 180,E1 -26678.715,E2 -26678.715} C_VEL
LIN {X 0,Y 137.726,Z 523.134,A -85,B 0,C 180,E1 -26680.057,E2 -26680.057} C_VEL
LIN {X 0,Y 135.577,Z 525.009,A -85,B 0,C 180,E1 -26681.269,E2 -26681.269} C_VEL
LIN {X 0,Y 128.26,Z 530.18,A -85,B 0,C 180,E1 -26684.577,E2 -26684.577} C_VEL
LIN {X 0,Y 121.52,Z 534.308,A -85,B 0,C 180,E1 -26688.313,E2 -26688.313} C_VEL
LIN {X 0,Y 115.519,Z 537.501,A -85,B 0,C 180,E1 -26692.529,E2 -26692.529} C_VEL
LIN {X 0,Y 108.642,Z 540.454,A -85,B 0,C 180,E1 -26698.836,E2 -26698.836} C_VEL
LIN {X 0,Y 103.265,Z 541.957,A -85,B 0,C 180,E1 -26705.901,E2 -26705.901} C_VEL
LIN {X 0,Y 99.893,Z 542.017,A -85,B 0,C 180,E1 -26713.657,E2 -26713.657} C_VEL
LIN {X 0,Y 98.373,Z 540.667,A -85,B 0,C 180,E1 -26721.787,E2 -26721.787} C_VEL
LIN {X 0,Y 98.405,Z 538.198,A -85,B 0,C 180,E1 -26729.082,E2 -26729.082} C_VEL
LIN {X 0,Y 98.39,Z 534.36,A -85,B 0,C 180,E1 -26736.152,E2 -26736.152} C_VEL
LIN {X 0,Y 99.059,Z 529.814,A -85,B 0,C 180,E1 -26742.29,E2 -26742.29} C_VEL
LIN {X 0,Y 100.938,Z 522.9,A -85,B 0,C 180,E1 -26749.314,E2 -26749.314} C_VEL
LIN {X 0,Y 103.661,Z 515.393,A -85,B 0,C 180,E1 -26755.072,E2 -26755.072} C_VEL
LIN {X 0,Y 106.539,Z 507.696,A -85,B 0,C 180,E1 -26759.655,E2 -26759.655} C_VEL
LIN {X 0,Y 109.752,Z 499.163,A -85,B 0,C 180,E1 -26763.647,E2 -26763.647} C_VEL
LIN {X 0,Y 110.513,Z 489.518,A -85,B 0,C 180,E1 -26767.743,E2 -26767.743} C_VEL
LIN {X 0,Y 110.95,Z 477.936,A -85,B 0,C 180,E1 -26771.894,E2 -26771.894} C_VEL
LIN {X 0,Y 110.691,Z 465.391,A -85,B 0,C 180,E1 -26775.7,E2 -26775.7} C_VEL
LIN {X 0,Y 109.665,Z 460.023,A -85,B 0,C 180,E1 -26777.381,E2 -26777.381} C_VEL
LIN {X 0,Y 105.895,Z 449.115,A -85,B 0,C 180,E1 -26781.145,E2 -26781.145} C_VEL
LIN {X 0,Y 102.995,Z 442.112,A -85,B 0,C 180,E1 -26783.643,E2 -26783.643} C_VEL
LIN {X 0,Y 101.304,Z 439.749,A -85,B 0,C 180,E1 -26784.782,E2 -26784.782} C_VEL
LIN {X 0,Y 100.768,Z 437.923,A -85,B 0,C 180,E1 -26785.329,E2 -26785.329} C_VEL
LIN {X 0,Y 100.672,Z 437.933,A -85,B 0,C 180,E1 -26790.746,E2 -26790.746} C_VEL
LIN {X 0,Y 100.789,Z 437.919,A -85,B 0,C 180,E1 -26795.267,E2 -26795.267} C_VEL
LIN {X 0,Y 100.821,Z 437.925,A -85,B 0,C 180,E1 -26799.602,E2 -26799.602} C_VEL
LIN {X 0,Y 101.191,Z 437.872,A -85,B 0,C 180,E1 -26807.973,E2 -26807.973} C_VEL
LIN {X 0,Y 101.27,Z 437.869,A -85,B 0,C 180,E1 -26812.021,E2 -26812.021} C_VEL
LIN {X 0,Y 101.871,Z 437.792,A -85,B 0,C 180,E1 -26820,E2 -26820} C_VEL
LIN {X 0,Y 101.274,Z 437.865,A -85,B 0,C 180,E1 -26827.978,E2 -26827.978} C_VEL
LIN {X 0,Y 101.13,Z 437.871,A -85,B 0,C 180,E1 -26833.357,E2 -26833.357} C_VEL
LIN {X 0,Y 100.745,Z 437.902,A -85,B 0,C 180,E1 -26841.833,E2 -26841.833} C_VEL
LIN {X 0,Y 100.777,Z 437.928,A -85,B 0,C 180,E1 -26844.958,E2 -26844.958} C_VEL
LIN {X 0,Y 100.698,Z 437.912,A -85,B 0,C 180,E1 -26853.12,E2 -26853.12} C_VEL
LIN {X 0,Y 100.63,Z 437.928,A -85,B 0,C 180,E1 -26858.991,E2 -26858.991} C_VEL
LIN {X 0,Y 99.963,Z 438.03,A -85,B 0,C 180,E1 -26862.33,E2 -26862.33} C_VEL
LIN {X 0,Y 98.387,Z 438.228,A -85,B 0,C 180,E1 -26865.637,E2 -26865.637} C_VEL
LIN {X 0,Y 93.867,Z 438.784,A -85,B 0,C 180,E1 -26874.895,E2 -26874.895} C_VEL
LIN {X 0,Y 93.572,Z 438.825,A -85,B 0,C 180,E1 -26877.364,E2 -26877.364} C_VEL
LIN {X 0,Y 93.671,Z 438.8,A -85,B 0,C 180,E1 -26884.203,E2 -26884.203} C_VEL
LIN {X 0,Y 93.697,Z 438.815,A -85,B 0,C 180,E1 -26887.972,E2 -26887.972} C_VEL
LIN {X 0,Y 93.974,Z 438.782,A -85,B 0,C 180,E1 -26895.489,E2 -26895.489} C_VEL
LIN {X 0,Y 95.19,Z 441.735,A -85,B 0,C 180,E1 -26896.879,E2 -26896.879} C_VEL
LIN {X 0,Y 96.456,Z 443.41,A -85,B 0,C 180,E1 -26897.907,E2 -26897.907} C_VEL
LIN {X 0,Y 102.155,Z 454.681,A -85,B 0,C 180,E1 -26903.37,E2 -26903.37} C_VEL
LIN {X 0,Y 104.112,Z 459.842,A -85,B 0,C 180,E1 -26905.643,E2 -26905.643} C_VEL
LIN {X 0,Y 105.695,Z 466.42,A -85,B 0,C 180,E1 -26908.316,E2 -26908.316} C_VEL
LIN {X 0,Y 106.4,Z 476.523,A -85,B 0,C 180,E1 -26912.223,E2 -26912.223} C_VEL
LIN {X 0,Y 106.578,Z 484.592,A -85,B 0,C 180,E1 -26915.677,E2 -26915.677} C_VEL
LIN {X 0,Y 102.628,Z 494.747,A -85,B 0,C 180,E1 -26919.856,E2 -26919.856} C_VEL
LIN {X 0,Y 99.191,Z 503.172,A -85,B 0,C 180,E1 -26924.355,E2 -26924.355} C_VEL
LIN {X 0,Y 95.875,Z 511.47,A -85,B 0,C 180,E1 -26930.104,E2 -26930.104} C_VEL
LIN {X 0,Y 93.152,Z 518.898,A -85,B 0,C 180,E1 -26936.914,E2 -26936.914} C_VEL
LIN {X 0,Y 91.416,Z 524.669,A -85,B 0,C 180,E1 -26943.869,E2 -26943.869} C_VEL
LIN {X 0,Y 90.476,Z 529.454,A -85,B 0,C 180,E1 -26951.594,E2 -26951.594} C_VEL
LIN {X 0,Y 90.532,Z 531.391,A -85,B 0,C 180,E1 -26955.68,E2 -26955.68} C_VEL
LIN {X 0,Y 91.397,Z 533.765,A -85,B 0,C 180,E1 -26962.037,E2 -26962.037} C_VEL
LIN {X 0,Y 93.172,Z 535.291,A -85,B 0,C 180,E1 -26968.129,E2 -26968.129} C_VEL
LIN {X 0,Y 95.838,Z 536.094,A -85,B 0,C 180,E1 -26973.897,E2 -26973.897} C_VEL
LIN {X 0,Y 99.257,Z 536.203,A -85,B 0,C 180,E1 -26979.266,E2 -26979.266} C_VEL
LIN {X 0,Y 103.438,Z 535.582,A -85,B 0,C 180,E1 -26984.23,E2 -26984.23} C_VEL
LIN {X 0,Y 108.295,Z 534.314,A -85,B 0,C 180,E1 -26988.774,E2 -26988.774} C_VEL
LIN {X 0,Y 116.868,Z 531.021,A -85,B 0,C 180,E1 -26994.827,E2 -26994.827} C_VEL
LIN {X 0,Y 126.629,Z 525.954,A -85,B 0,C 180,E1 -27000,E2 -27000} C_VEL
LIN {X 0,Y 135.543,Z 520.206,A -85,B 0,C 180,E1 -27003.716,E2 -27003.716} C_VEL
LIN {X 0,Y 137.081,Z 519.069,A -85,B 0,C 180,E1 -27004.411,E2 -27004.411} C_VEL
LIN {X 0,Y 138.006,Z 517.906,A -85,B 0,C 180,E1 -27005.846,E2 -27005.846} C_VEL
LIN {X 0,Y 139.063,Z 516.18,A -85,B 0,C 180,E1 -27008.721,E2 -27008.721} C_VEL
LIN {X 0,Y 139.615,Z 514.951,A -85,B 0,C 180,E1 -27011.616,E2 -27011.616} C_VEL
LIN {X 0,Y 139.816,Z 514.201,A -85,B 0,C 180,E1 -27014.556,E2 -27014.556} C_VEL
LIN {X 0,Y 139.747,Z 513.976,A -85,B 0,C 180,E1 -27017.563,E2 -27017.563} C_VEL
LIN {X 0,Y 139.461,Z 514.198,A -85,B 0,C 180,E1 -27020.656,E2 -27020.656} C_VEL
LIN {X 0,Y 139.192,Z 515.038,A -85,B 0,C 180,E1 -27024.658,E2 -27024.658} C_VEL
LIN {X 0,Y 138.786,Z 515.956,A -85,B 0,C 180,E1 -27027.114,E2 -27027.114} C_VEL
LIN {X 0,Y 138.215,Z 517.631,A -85,B 0,C 180,E1 -27030.563,E2 -27030.563} C_VEL
LIN {X 0,Y 137.75,Z 518.762,A -85,B 0,C 180,E1 -27032.392,E2 -27032.392} C_VEL
LIN {X 0,Y 136.731,Z 520.526,A -85,B 0,C 180,E1 -27034.677,E2 -27034.677} C_VEL
LIN {X 0,Y 135.133,Z 522.344,A -85,B 0,C 180,E1 -27036.283,E2 -27036.283} C_VEL
LIN {X 0,Y 133.183,Z 524.126,A -85,B 0,C 180,E1 -27037.672,E2 -27037.672} C_VEL
LIN {X 0,Y 131.009,Z 525.915,A -85,B 0,C 180,E1 -27038.938,E2 -27038.938} C_VEL
LIN {X 0,Y 120.96,Z 532.225,A -85,B 0,C 180,E1 -27043.427,E2 -27043.427} C_VEL
LIN {X 0,Y 114.104,Z 535.835,A -85,B 0,C 180,E1 -27047.352,E2 -27047.352} C_VEL
LIN {X 0,Y 106.156,Z 539.296,A -85,B 0,C 180,E1 -27053.43,E2 -27053.43} C_VEL
LIN {X 0,Y 99.532,Z 541.267,A -85,B 0,C 180,E1 -27060.38,E2 -27060.38} C_VEL
LIN {X 0,Y 94.644,Z 541.835,A -85,B 0,C 180,E1 -27068.207,E2 -27068.207} C_VEL
LIN {X 0,Y 91.971,Z 541.031,A -85,B 0,C 180,E1 -27076.749,E2 -27076.749} C_VEL
LIN {X 0,Y 91.215,Z 538.724,A -85,B 0,C 180,E1 -27085.583,E2 -27085.583} C_VEL
LIN {X 0,Y 91.368,Z 536.76,A -85,B 0,C 180,E1 -27090.447,E2 -27090.447} C_VEL
LIN {X 0,Y 91.364,Z 533.37,A -85,B 0,C 180,E1 -27096.627,E2 -27096.627} C_VEL
LIN {X 0,Y 92.124,Z 528.627,A -85,B 0,C 180,E1 -27103.232,E2 -27103.232} C_VEL
LIN {X 0,Y 93.862,Z 522.606,A -85,B 0,C 180,E1 -27109.692,E2 -27109.692} C_VEL
LIN {X 0,Y 96.682,Z 515.122,A -85,B 0,C 180,E1 -27115.86,E2 -27115.86} C_VEL
LIN {X 0,Y 99.717,Z 507.457,A -85,B 0,C 180,E1 -27120.731,E2 -27120.731} C_VEL
LIN {X 0,Y 102.611,Z 500.492,A -85,B 0,C 180,E1 -27124.234,E2 -27124.234} C_VEL
LIN {X 0,Y 103.272,Z 496.523,A -85,B 0,C 180,E1 -27126.124,E2 -27126.124} C_VEL
LIN {X 0,Y 104.077,Z 486.327,A -85,B 0,C 180,E1 -27130.539,E2 -27130.539} C_VEL
LIN {X 0,Y 104.502,Z 475.01,A -85,B 0,C 180,E1 -27134.666,E2 -27134.666} C_VEL
LIN {X 0,Y 104.326,Z 465.786,A -85,B 0,C 180,E1 -27137.649,E2 -27137.649} C_VEL
LIN {X 0,Y 102.242,Z 458.111,A -85,B 0,C 180,E1 -27140.516,E2 -27140.516} C_VEL
LIN {X 0,Y 98.571,Z 448.101,A -85,B 0,C 180,E1 -27144.441,E2 -27144.441} C_VEL
LIN {X 0,Y 97.315,Z 445.863,A -85,B 0,C 180,E1 -27145.502,E2 -27145.502} C_VEL
LIN {X 0,Y 95.587,Z 442.793,A -85,B 0,C 180,E1 -27146.992,E2 -27146.992} C_VEL
LIN {X 0,Y 94.015,Z 440.339,A -85,B 0,C 180,E1 -27148.3,E2 -27148.3} C_VEL
LIN {X 0,Y 93.62,Z 438.825,A -85,B 0,C 180,E1 -27148.928,E2 -27148.928} C_VEL
LIN {X 0,Y 93.672,Z 438.798,A -85,B 0,C 180,E1 -27154.204,E2 -27154.204} C_VEL
LIN {X 0,Y 93.698,Z 438.814,A -85,B 0,C 180,E1 -27157.973,E2 -27157.973} C_VEL
LIN {X 0,Y 94.094,Z 438.758,A -85,B 0,C 180,E1 -27167.051,E2 -27167.051} C_VEL
LIN {X 0,Y 94.203,Z 438.749,A -85,B 0,C 180,E1 -27171.419,E2 -27171.419} C_VEL
LIN {X 0,Y 94.797,Z 438.673,A -85,B 0,C 180,E1 -27180,E2 -27180} C_VEL
LIN {X 0,Y 94.207,Z 438.747,A -85,B 0,C 180,E1 -27188.58,E2 -27188.58} C_VEL
LIN {X 0,Y 94.048,Z 438.748,A -85,B 0,C 180,E1 -27193.716,E2 -27193.716} C_VEL
LIN {X 0,Y 93.695,Z 438.791,A -85,B 0,C 180,E1 -27202.027,E2 -27202.027} C_VEL
LIN {X 0,Y 93.625,Z 438.823,A -85,B 0,C 180,E1 -27206.768,E2 -27206.768} C_VEL
LIN {X 0,Y 93.593,Z 438.787,A -85,B 0,C 180,E1 -27214.308,E2 -27214.308} C_VEL
LIN {X 0,Y 93.534,Z 438.831,A -85,B 0,C 180,E1 -27222.551,E2 -27222.551} C_VEL
LIN {X 0,Y 93.544,Z 438.81,A -85,B 0,C 180,E1 -27228.703,E2 -27228.703} C_VEL
LIN {X 0,Y 93.6,Z 438.822,A -85,B 0,C 180,E1 -27235.684,E2 -27235.684} C_VEL
LIN {X 0,Y 93.572,Z 438.825,A -85,B 0,C 180,E1 -27237.364,E2 -27237.364} C_VEL
LIN {X 0,Y 92.893,Z 438.912,A -85,B 0,C 180,E1 -27239.739,E2 -27239.739} C_VEL
LIN {X 0,Y 90.03,Z 439.261,A -85,B 0,C 180,E1 -27243.516,E2 -27243.516} C_VEL
LIN {X 0,Y 87.168,Z 439.628,A -85,B 0,C 180,E1 -27247.534,E2 -27247.534} C_VEL
LIN {X 0,Y 86.591,Z 439.682,A -85,B 0,C 180,E1 -27250.177,E2 -27250.177} C_VEL
LIN {X 0,Y 86.674,Z 439.711,A -85,B 0,C 180,E1 -27251.325,E2 -27251.325} C_VEL
LIN {X 0,Y 87.676,Z 442.37,A -85,B 0,C 180,E1 -27252.68,E2 -27252.68} C_VEL
LIN {X 0,Y 89.725,Z 445.146,A -85,B 0,C 180,E1 -27254.672,E2 -27254.672} C_VEL
LIN {X 0,Y 92.276,Z 449.707,A -85,B 0,C 180,E1 -27257.405,E2 -27257.405} C_VEL
LIN {X 0,Y 96.487,Z 458.412,A -85,B 0,C 180,E1 -27262.148,E2 -27262.148} C_VEL
LIN {X 0,Y 98.19,Z 463.095,A -85,B 0,C 180,E1 -27264.43,E2 -27264.43} C_VEL
LIN {X 0,Y 99.51,Z 469.361,A -85,B 0,C 180,E1 -27267.181,E2 -27267.181} C_VEL
LIN {X 0,Y 99.91,Z 479.852,A -85,B 0,C 180,E1 -27271.686,E2 -27271.686} C_VEL
LIN {X 0,Y 99.928,Z 484.843,A -85,B 0,C 180,E1 -27274.031,E2 -27274.031} C_VEL
LIN {X 0,Y 96.78,Z 492.952,A -85,B 0,C 180,E1 -27277.473,E2 -27277.473} C_VEL
LIN {X 0,Y 92.329,Z 503.358,A -85,B 0,C 180,E1 -27283.199,E2 -27283.199} C_VEL
LIN {X 0,Y 88.63,Z 512.199,A -85,B 0,C 180,E1 -27289.812,E2 -27289.812} C_VEL
LIN {X 0,Y 85.712,Z 520.01,A -85,B 0,C 180,E1 -27297.741,E2 -27297.741} C_VEL
LIN {X 0,Y 84.333,Z 524.397,A -85,B 0,C 180,E1 -27303.555,E2 -27303.555} C_VEL
LIN {X 0,Y 83.37,Z 529.541,A -85,B 0,C 180,E1 -27312.404,E2 -27312.404} C_VEL
LIN {X 0,Y 83.739,Z 532.367,A -85,B 0,C 180,E1 -27319.052,E2 -27319.052} C_VEL
LIN {X 0,Y 85.109,Z 534.473,A -85,B 0,C 180,E1 -27325.662,E2 -27325.662} C_VEL
LIN {X 0,Y 87.485,Z 535.867,A -85,B 0,C 180,E1 -27332.084,E2 -27332.084} C_VEL
LIN {X 0,Y 90.832,Z 536.489,A -85,B 0,C 180,E1 -27338.194,E2 -27338.194} C_VEL
LIN {X 0,Y 95.111,Z 536.391,A -85,B 0,C 180,E1 -27343.857,E2 -27343.857} C_VEL
LIN {X 0,Y 100.223,Z 535.572,A -85,B 0,C 180,E1 -27349.022,E2 -27349.022} C_VEL
LIN {X 0,Y 106.073,Z 533.973,A -85,B 0,C 180,E1 -27353.621,E2 -27353.621} C_VEL
LIN {X 0,Y 112.535,Z 531.607,A -85,B 0,C 180,E1 -27357.7,E2 -27357.7} C_VEL
LIN {X 0,Y 121.692,Z 527.349,A -85,B 0,C 180,E1 -27362.277,E2 -27362.277} C_VEL
LIN {X 0,Y 131.467,Z 521.569,A -85,B 0,C 180,E1 -27366.138,E2 -27366.138} C_VEL
LIN {X 0,Y 133.009,Z 519.863,A -85,B 0,C 180,E1 -27369.121,E2 -27369.121} C_VEL
LIN {X 0,Y 133.688,Z 518.741,A -85,B 0,C 180,E1 -27372.139,E2 -27372.139} C_VEL
LIN {X 0,Y 133.928,Z 518.144,A -85,B 0,C 180,E1 -27375.212,E2 -27375.212} C_VEL
LIN {X 0,Y 133.736,Z 518.135,A -85,B 0,C 180,E1 -27378.933,E2 -27378.933} C_VEL
LIN {X 0,Y 133.525,Z 518.435,A -85,B 0,C 180,E1 -27381.62,E2 -27381.62} C_VEL
LIN {X 0,Y 132.989,Z 519.542,A -85,B 0,C 180,E1 -27386.056,E2 -27386.056} C_VEL
LIN {X 0,Y 132.505,Z 520.535,A -85,B 0,C 180,E1 -27388.513,E2 -27388.513} C_VEL
LIN {X 0,Y 131.815,Z 522.014,A -85,B 0,C 180,E1 -27391.455,E2 -27391.455} C_VEL
LIN {X 0,Y 130.939,Z 523.185,A -85,B 0,C 180,E1 -27393.225,E2 -27393.225} C_VEL
LIN {X 0,Y 128.839,Z 525.137,A -85,B 0,C 180,E1 -27395.095,E2 -27395.095} C_VEL
LIN {X 0,Y 126.643,Z 526.778,A -85,B 0,C 180,E1 -27396.424,E2 -27396.424} C_VEL
LIN {X 0,Y 118.773,Z 531.438,A -85,B 0,C 180,E1 -27399.718,E2 -27399.718} C_VEL
LIN {X 0,Y 108.992,Z 536.19,A -85,B 0,C 180,E1 -27404.825,E2 -27404.825} C_VEL
LIN {X 0,Y 100.529,Z 539.37,A -85,B 0,C 180,E1 -27411.012,E2 -27411.012} C_VEL
LIN {X 0,Y 93.409,Z 541.13,A -85,B 0,C 180,E1 -27418.221,E2 -27418.221} C_VEL
LIN {X 0,Y 88.064,Z 541.513,A -85,B 0,C 180,E1 -27426.485,E2 -27426.485} C_VEL
LIN {X 0,Y 85.075,Z 540.464,A -85,B 0,C 180,E1 -27435.653,E2 -27435.653} C_VEL
LIN {X 0,Y 84.16,Z 537.97,A -85,B 0,C 180,E1 -27445.212,E2 -27445.212} C_VEL
LIN {X 0,Y 84.337,Z 536.14,A -85,B 0,C 180,E1 -27450.002,E2 -27450.002} C_VEL
LIN {X 0,Y 84.323,Z 532.378,A -85,B 0,C 180,E1 -27457.184,E2 -27457.184} C_VEL
LIN {X 0,Y 85.228,Z 527.443,A -85,B 0,C 180,E1 -27464.325,E2 -27464.325} C_VEL
LIN {X 0,Y 87.202,Z 521.193,A -85,B 0,C 180,E1 -27471.266,E2 -27471.266} C_VEL
LIN {X 0,Y 90.339,Z 513.378,A -85,B 0,C 180,E1 -27477.827,E2 -27477.827} C_VEL
LIN {X 0,Y 94.464,Z 503.682,A -85,B 0,C 180,E1 -27483.918,E2 -27483.918} C_VEL
LIN {X 0,Y 96.042,Z 499.893,A -85,B 0,C 180,E1 -27485.833,E2 -27485.833} C_VEL
LIN {X 0,Y 97.084,Z 491.423,A -85,B 0,C 180,E1 -27490.033,E2 -27490.033} C_VEL
LIN {X 0,Y 97.941,Z 480.922,A -85,B 0,C 180,E1 -27494.503,E2 -27494.503} C_VEL
LIN {X 0,Y 98.203,Z 468.809,A -85,B 0,C 180,E1 -27498.913,E2 -27498.913} C_VEL
LIN {X 0,Y 96.742,Z 462.354,A -85,B 0,C 180,E1 -27501.534,E2 -27501.534} C_VEL
LIN {X 0,Y 93.602,Z 452.779,A -85,B 0,C 180,E1 -27505.684,E2 -27505.684} C_VEL
LIN {X 0,Y 90.79,Z 447.538,A -85,B 0,C 180,E1 -27508.535,E2 -27508.535} C_VEL
LIN {X 0,Y 88.731,Z 443.927,A -85,B 0,C 180,E1 -27510.651,E2 -27510.651} C_VEL
LIN {X 0,Y 87.019,Z 441.417,A -85,B 0,C 180,E1 -27512.28,E2 -27512.28} C_VEL
LIN {X 0,Y 86.585,Z 439.677,A -85,B 0,C 180,E1 -27513.056,E2 -27513.056} C_VEL
LIN {X 0,Y 86.651,Z 439.684,A -85,B 0,C 180,E1 -27521.069,E2 -27521.069} C_VEL
LIN {X 0,Y 86.972,Z 439.65,A -85,B 0,C 180,E1 -27525.97,E2 -27525.97} C_VEL
LIN {X 0,Y 87.111,Z 439.63,A -85,B 0,C 180,E1 -27530.714,E2 -27530.714} C_VEL
LIN {X 0,Y 87.725,Z 439.554,A -85,B 0,C 180,E1 -27540,E2 -27540} C_VEL
LIN {X 0,Y 87.115,Z 439.63,A -85,B 0,C 180,E1 -27549.285,E2 -27549.285} C_VEL
LIN {X 0,Y 86.953,Z 439.627,A -85,B 0,C 180,E1 -27554.087,E2 -27554.087} C_VEL
LIN {X 0,Y 86.589,Z 439.689,A -85,B 0,C 180,E1 -27563.942,E2 -27563.942} C_VEL
LIN {X 0,Y 86.48,Z 439.709,A -85,B 0,C 180,E1 -27569.183,E2 -27569.183} C_VEL
LIN {X 0,Y 86.511,Z 439.664,A -85,B 0,C 180,E1 -27575.668,E2 -27575.668} C_VEL
LIN {X 0,Y 86.477,Z 439.712,A -85,B 0,C 180,E1 -27582.991,E2 -27582.991} C_VEL
LIN {X 0,Y 86.466,Z 439.686,A -85,B 0,C 180,E1 -27589.438,E2 -27589.438} C_VEL
LIN {X 0,Y 86.544,Z 439.698,A -85,B 0,C 180,E1 -27595.356,E2 -27595.356} C_VEL
LIN {X 0,Y 86.587,Z 439.679,A -85,B 0,C 180,E1 -27603.232,E2 -27603.232} C_VEL
LIN {X 0,Y 86.591,Z 439.682,A -85,B 0,C 180,E1 -27610.177,E2 -27610.177} C_VEL
LIN {X 0,Y 87.384,Z 440.245,A -85,B 0,C 180,E1 -27611.845,E2 -27611.845} C_VEL
LIN {X 0,Y 89.231,Z 442.173,A -85,B 0,C 180,E1 -27613.593,E2 -27613.593} C_VEL
LIN {X 0,Y 90.817,Z 445.798,A -85,B 0,C 180,E1 -27615.485,E2 -27615.485} C_VEL
LIN {X 0,Y 91.684,Z 451.235,A -85,B 0,C 180,E1 -27617.396,E2 -27617.396} C_VEL
LIN {X 0,Y 91.552,Z 457.284,A -85,B 0,C 180,E1 -27619.253,E2 -27619.253} C_VEL
LIN {X 0,Y 91.512,Z 462.983,A -85,B 0,C 180,E1 -27621.463,E2 -27621.463} C_VEL
LIN {X 0,Y 91.836,Z 464.716,A -85,B 0,C 180,E1 -27622.314,E2 -27622.314} C_VEL
LIN {X 0,Y 93.232,Z 471.454,A -85,B 0,C 180,E1 -27625.675,E2 -27625.675} C_VEL
LIN {X 0,Y 93.409,Z 480.762,A -85,B 0,C 180,E1 -27629.998,E2 -27629.998} C_VEL
LIN {X 0,Y 93.211,Z 486.115,A -85,B 0,C 180,E1 -27632.674,E2 -27632.674} C_VEL
LIN {X 0,Y 88.88,Z 496.136,A -85,B 0,C 180,E1 -27637.381,E2 -27637.381} C_VEL
LIN {X 0,Y 85.013,Z 504.644,A -85,B 0,C 180,E1 -27642.684,E2 -27642.684} C_VEL
LIN {X 0,Y 81.675,Z 512.155,A -85,B 0,C 180,E1 -27648.822,E2 -27648.822} C_VEL
LIN {X 0,Y 78.751,Z 519.54,A -85,B 0,C 180,E1 -27656.82,E2 -27656.82} C_VEL
LIN {X 0,Y 76.974,Z 525.068,A -85,B 0,C 180,E1 -27664.741,E2 -27664.741} C_VEL
LIN {X 0,Y 76.299,Z 529.225,A -85,B 0,C 180,E1 -27672.533,E2 -27672.533} C_VEL
LIN {X 0,Y 76.769,Z 532.334,A -85,B 0,C 180,E1 -27680.147,E2 -27680.147} C_VEL
LIN {X 0,Y 78.4,Z 534.58,A -85,B 0,C 180,E1 -27687.463,E2 -27687.463} C_VEL
LIN {X 0,Y 81.097,Z 536.026,A -85,B 0,C 180,E1 -27694.323,E2 -27694.323} C_VEL
LIN {X 0,Y 84.706,Z 536.74,A -85,B 0,C 180,E1 -27700.618,E2 -27700.618} C_VEL
LIN {X 0,Y 89.211,Z 536.798,A -85,B 0,C 180,E1 -27706.33,E2 -27706.33} C_VEL
LIN {X 0,Y 94.461,Z 536.14,A -85,B 0,C 180,E1 -27711.443,E2 -27711.443} C_VEL
LIN {X 0,Y 100.447,Z 534.807,A -85,B 0,C 180,E1 -27715.988,E2 -27715.988} C_VEL
LIN {X 0,Y 110.015,Z 531.654,A -85,B 0,C 180,E1 -27721.552,E2 -27721.552} C_VEL
LIN {X 0,Y 120.139,Z 527.098,A -85,B 0,C 180,E1 -27726.039,E2 -27726.039} C_VEL
LIN {X 0,Y 125.65,Z 524.103,A -85,B 0,C 180,E1 -27728.038,E2 -27728.038} C_VEL
LIN {X 0,Y 126.719,Z 523.252,A -85,B 0,C 180,E1 -27729.578,E2 -27729.578} C_VEL
LIN {X 0,Y 127.583,Z 522.246,A -85,B 0,C 180,E1 -27732.729,E2 -27732.729} C_VEL
LIN {X 0,Y 127.816,Z 521.818,A -85,B 0,C 180,E1 -27735.958,E2 -27735.958} C_VEL
LIN {X 0,Y 127.53,Z 522,A -85,B 0,C 180,E1 -27740.477,E2 -27740.477} C_VEL
LIN {X 0,Y 127.29,Z 522.384,A -85,B 0,C 180,E1 -27742.736,E2 -27742.736} C_VEL
LIN {X 0,Y 126.513,Z 523.661,A -85,B 0,C 180,E1 -27747.278,E2 -27747.278} C_VEL
LIN {X 0,Y 125.787,Z 524.895,A -85,B 0,C 180,E1 -27750.189,E2 -27750.189} C_VEL
LIN {X 0,Y 124.577,Z 526.134,A -85,B 0,C 180,E1 -27752.2,E2 -27752.2} C_VEL
LIN {X 0,Y 122.5,Z 527.663,A -85,B 0,C 180,E1 -27753.71,E2 -27753.71} C_VEL
LIN {X 0,Y 114.382,Z 532.057,A -85,B 0,C 180,E1 -27756.991,E2 -27756.991} C_VEL
LIN {X 0,Y 104.107,Z 536.496,A -85,B 0,C 180,E1 -27762.051,E2 -27762.051} C_VEL
LIN {X 0,Y 95.105,Z 539.433,A -85,B 0,C 180,E1 -27768.314,E2 -27768.314} C_VEL
LIN {X 0,Y 87.427,Z 540.989,A -85,B 0,C 180,E1 -27775.759,E2 -27775.759} C_VEL
LIN {X 0,Y 81.583,Z 541.107,A -85,B 0,C 180,E1 -27784.489,E2 -27784.489} C_VEL
LIN {X 0,Y 78.222,Z 539.878,A -85,B 0,C 180,E1 -27794.365,E2 -27794.365} C_VEL
LIN {X 0,Y 77.126,Z 537.202,A -85,B 0,C 180,E1 -27804.774,E2 -27804.774} C_VEL
LIN {X 0,Y 77.287,Z 535.223,A -85,B 0,C 180,E1 -27810.002,E2 -27810.002} C_VEL
LIN {X 0,Y 77.31,Z 531.272,A -85,B 0,C 180,E1 -27817.839,E2 -27817.839} C_VEL
LIN {X 0,Y 78.376,Z 526.129,A -85,B 0,C 180,E1 -27825.607,E2 -27825.607} C_VEL
LIN {X 0,Y 80.627,Z 519.64,A -85,B 0,C 180,E1 -27833.097,E2 -27833.097} C_VEL
LIN {X 0,Y 84.109,Z 511.596,A -85,B 0,C 180,E1 -27840.091,E2 -27840.091} C_VEL
LIN {X 0,Y 87.816,Z 503.383,A -85,B 0,C 180,E1 -27845.468,E2 -27845.468} C_VEL
LIN {X 0,Y 89.375,Z 499.843,A -85,B 0,C 180,E1 -27847.365,E2 -27847.365} C_VEL
LIN {X 0,Y 90.57,Z 491.114,A -85,B 0,C 180,E1 -27852.013,E2 -27852.013} C_VEL
LIN {X 0,Y 91.614,Z 480.307,A -85,B 0,C 180,E1 -27856.9,E2 -27856.9} C_VEL
LIN {X 0,Y 91.994,Z 470.43,A -85,B 0,C 180,E1 -27860.79,E2 -27860.79} C_VEL
LIN {X 0,Y 90.238,Z 463.083,A -85,B 0,C 180,E1 -27864.214,E2 -27864.214} C_VEL
LIN {X 0,Y 88.186,Z 456.439,A -85,B 0,C 180,E1 -27867.494,E2 -27867.494} C_VEL
LIN {X 0,Y 84.047,Z 448.83,A -85,B 0,C 180,E1 -27872.354,E2 -27872.354} C_VEL
LIN {X 0,Y 81.931,Z 445.037,A -85,B 0,C 180,E1 -27874.941,E2 -27874.941} C_VEL
LIN {X 0,Y 80.007,Z 442.445,A -85,B 0,C 180,E1 -27877.228,E2 -27877.228} C_VEL
LIN {X 0,Y 79.513,Z 440.582,A -85,B 0,C 180,E1 -27878.276,E2 -27878.276} C_VEL
LIN {X 0,Y 79.844,Z 440.539,A -85,B 0,C 180,E1 -27885.526,E2 -27885.526} C_VEL
LIN {X 0,Y 79.996,Z 440.512,A -85,B 0,C 180,E1 -27889.88,E2 -27889.88} C_VEL
LIN {X 0,Y 80.652,Z 440.435,A -85,B 0,C 180,E1 -27900,E2 -27900} C_VEL
LIN {X 0,Y 79.999,Z 440.516,A -85,B 0,C 180,E1 -27910.119,E2 -27910.119} C_VEL
LIN {X 0,Y 79.765,Z 440.508,A -85,B 0,C 180,E1 -27915.327,E2 -27915.327} C_VEL
LIN {X 0,Y 79.516,Z 440.539,A -85,B 0,C 180,E1 -27920.704,E2 -27920.704} C_VEL
LIN {X 0,Y 79.485,Z 440.584,A -85,B 0,C 180,E1 -27927.845,E2 -27927.845} C_VEL
LIN {X 0,Y 79.382,Z 440.571,A -85,B 0,C 180,E1 -27932.086,E2 -27932.086} C_VEL
LIN {X 0,Y 79.368,Z 440.563,A -85,B 0,C 180,E1 -27938.305,E2 -27938.305} C_VEL
LIN {X 0,Y 79.388,Z 440.594,A -85,B 0,C 180,E1 -27945.09,E2 -27945.09} C_VEL
LIN {X 0,Y 79.394,Z 440.567,A -85,B 0,C 180,E1 -27952.814,E2 -27952.814} C_VEL
LIN {X 0,Y 79.386,Z 440.597,A -85,B 0,C 180,E1 -27957.913,E2 -27957.913} C_VEL
LIN {X 0,Y 79.547,Z 440.563,A -85,B 0,C 180,E1 -27965.186,E2 -27965.186} C_VEL
LIN {X 0,Y 79.561,Z 440.7,A -85,B 0,C 180,E1 -27966.147,E2 -27966.147} C_VEL
LIN {X 0,Y 80.507,Z 443.421,A -85,B 0,C 180,E1 -27967.808,E2 -27967.808} C_VEL
LIN {X 0,Y 82.411,Z 445.735,A -85,B 0,C 180,E1 -27970.053,E2 -27970.053} C_VEL
LIN {X 0,Y 83.685,Z 448.181,A -85,B 0,C 180,E1 -27971.767,E2 -27971.767} C_VEL
LIN {X 0,Y 85.511,Z 450.935,A -85,B 0,C 180,E1 -27973.892,E2 -27973.892} C_VEL
LIN {X 0,Y 89.233,Z 458.391,A -85,B 0,C 180,E1 -27978.64,E2 -27978.64} C_VEL
LIN {X 0,Y 91.836,Z 464.716,A -85,B 0,C 180,E1 -27982.314,E2 -27982.314} C_VEL
LIN {X 0,Y 92.312,Z 467.892,A -85,B 0,C 180,E1 -27983.805,E2 -27983.805} C_VEL
LIN {X 0,Y 92.144,Z 471.272,A -85,B 0,C 180,E1 -27985.154,E2 -27985.154} C_VEL
LIN {X 0,Y 91.036,Z 476.39,A -85,B 0,C 180,E1 -27987.012,E2 -27987.012} C_VEL
LIN {X 0,Y 87.694,Z 484.743,A -85,B 0,C 180,E1 -27990.073,E2 -27990.073} C_VEL
LIN {X 0,Y 84.7,Z 491.079,A -85,B 0,C 180,E1 -27992.847,E2 -27992.847} C_VEL
LIN {X 0,Y 80.236,Z 500.487,A -85,B 0,C 180,E1 -27998.181,E2 -27998.181} C_VEL
LIN {X 0,Y 76.234,Z 508.942,A -85,B 0,C 180,E1 -28004.683,E2 -28004.683} C_VEL
LIN {X 0,Y 72.752,Z 516.704,A -85,B 0,C 180,E1 -28012.729,E2 -28012.729} C_VEL
LIN {X 0,Y 70.457,Z 522.911,A -85,B 0,C 180,E1 -28021.334,E2 -28021.334} C_VEL
LIN {X 0,Y 69.24,Z 528.135,A -85,B 0,C 180,E1 -28031.025,E2 -28031.025} C_VEL
LIN {X 0,Y 69.522,Z 531.453,A -85,B 0,C 180,E1 -28039.161,E2 -28039.161} C_VEL
LIN {X 0,Y 72.282,Z 534.992,A -85,B 0,C 180,E1 -28051.048,E2 -28051.048} C_VEL
LIN {X 0,Y 75.608,Z 536.421,A -85,B 0,C 180,E1 -28058.355,E2 -28058.355} C_VEL
LIN {X 0,Y 80.009,Z 537.085,A -85,B 0,C 180,E1 -28065.061,E2 -28065.061} C_VEL
LIN {X 0,Y 85.378,Z 537.049,A -85,B 0,C 180,E1 -28071.027,E2 -28071.027} C_VEL
LIN {X 0,Y 91.558,Z 536.298,A -85,B 0,C 180,E1 -28076.237,E2 -28076.237} C_VEL
LIN {X 0,Y 98.396,Z 534.77,A -85,B 0,C 180,E1 -28080.701,E2 -28080.701} C_VEL
LIN {X 0,Y 108.812,Z 531.429,A -85,B 0,C 180,E1 -28085.911,E2 -28085.911} C_VEL
LIN {X 0,Y 116.701,Z 528.074,A -85,B 0,C 180,E1 -28089.008,E2 -28089.008} C_VEL
LIN {X 0,Y 119.946,Z 526.478,A -85,B 0,C 180,E1 -28090.124,E2 -28090.124} C_VEL
LIN {X 0,Y 121.32,Z 525.462,A -85,B 0,C 180,E1 -28093.398,E2 -28093.398} C_VEL
LIN {X 0,Y 121.483,Z 525.216,A -85,B 0,C 180,E1 -28096.814,E2 -28096.814} C_VEL
LIN {X 0,Y 121.292,Z 525.382,A -85,B 0,C 180,E1 -28100.344,E2 -28100.344} C_VEL
LIN {X 0,Y 120.736,Z 526.086,A -85,B 0,C 180,E1 -28104.046,E2 -28104.046} C_VEL
LIN {X 0,Y 119.758,Z 527.366,A -85,B 0,C 180,E1 -28108.328,E2 -28108.328} C_VEL
LIN {X 0,Y 118.51,Z 528.52,A -85,B 0,C 180,E1 -28110.699,E2 -28110.699} C_VEL
LIN {X 0,Y 115.971,Z 529.96,A -85,B 0,C 180,E1 -28111.963,E2 -28111.963} C_VEL
LIN {X 0,Y 104.77,Z 534.889,A -85,B 0,C 180,E1 -28116.396,E2 -28116.396} C_VEL
LIN {X 0,Y 94.563,Z 538.325,A -85,B 0,C 180,E1 -28121.998,E2 -28121.998} C_VEL
LIN {X 0,Y 85.575,Z 540.299,A -85,B 0,C 180,E1 -28128.93,E2 -28128.93} C_VEL
LIN {X 0,Y 78.179,Z 540.899,A -85,B 0,C 180,E1 -28137.361,E2 -28137.361} C_VEL
LIN {X 0,Y 72.974,Z 540.148,A -85,B 0,C 180,E1 -28147.344,E2 -28147.344} C_VEL
LIN {X 0,Y 71.42,Z 539.264,A -85,B 0,C 180,E1 -28152.832,E2 -28152.832} C_VEL
LIN {X 0,Y 70.108,Z 536.343,A -85,B 0,C 180,E1 -28164.249,E2 -28164.249} C_VEL
LIN {X 0,Y 70.239,Z 534.276,A -85,B 0,C 180,E1 -28170.002,E2 -28170.002} C_VEL
LIN {X 0,Y 70.32,Z 530.124,A -85,B 0,C 180,E1 -28178.624,E2 -28178.624} C_VEL
LIN {X 0,Y 71.888,Z 523.758,A -85,B 0,C 180,E1 -28188.528,E2 -28188.528} C_VEL
LIN {X 0,Y 74.727,Z 516.749,A -85,B 0,C 180,E1 -28196.536,E2 -28196.536} C_VEL
LIN {X 0,Y 78.792,Z 508.041,A -85,B 0,C 180,E1 -28203.884,E2 -28203.884} C_VEL
LIN {X 0,Y 82.709,Z 499.78,A -85,B 0,C 180,E1 -28209.064,E2 -28209.064} C_VEL
LIN {X 0,Y 84.162,Z 490.507,A -85,B 0,C 180,E1 -28214.378,E2 -28214.378} C_VEL
LIN {X 0,Y 85.433,Z 479.62,A -85,B 0,C 180,E1 -28219.629,E2 -28219.629} C_VEL
LIN {X 0,Y 85.8,Z 472.217,A -85,B 0,C 180,E1 -28222.836,E2 -28222.836} C_VEL
LIN {X 0,Y 83.966,Z 464.129,A -85,B 0,C 180,E1 -28227.157,E2 -28227.157} C_VEL
LIN {X 0,Y 82.768,Z 460.185,A -85,B 0,C 180,E1 -28229.371,E2 -28229.371} C_VEL
LIN {X 0,Y 78.051,Z 450.975,A -85,B 0,C 180,E1 -28236.096,E2 -28236.096} C_VEL
LIN {X 0,Y 75.678,Z 447.039,A -85,B 0,C 180,E1 -28239.62,E2 -28239.62} C_VEL
LIN {X 0,Y 74.953,Z 445.996,A -85,B 0,C 180,E1 -28240.666,E2 -28240.666} C_VEL
LIN {X 0,Y 73.254,Z 443.642,A -85,B 0,C 180,E1 -28243.272,E2 -28243.272} C_VEL
LIN {X 0,Y 72.73,Z 441.426,A -85,B 0,C 180,E1 -28244.766,E2 -28244.766} C_VEL
LIN {X 0,Y 72.883,Z 441.395,A -85,B 0,C 180,E1 -28248.88,E2 -28248.88} C_VEL
LIN {X 0,Y 73.579,Z 441.316,A -85,B 0,C 180,E1 -28260,E2 -28260} C_VEL
LIN {X 0,Y 72.885,Z 441.399,A -85,B 0,C 180,E1 -28271.119,E2 -28271.119} C_VEL
LIN {X 0,Y 72.585,Z 441.392,A -85,B 0,C 180,E1 -28276.886,E2 -28276.886} C_VEL
LIN {X 0,Y 72.397,Z 441.445,A -85,B 0,C 180,E1 -28282.849,E2 -28282.849} C_VEL
LIN {X 0,Y 72.379,Z 441.465,A -85,B 0,C 180,E1 -28289.081,E2 -28289.081} C_VEL
LIN {X 0,Y 72.297,Z 441.432,A -85,B 0,C 180,E1 -28295.68,E2 -28295.68} C_VEL
LIN {X 0,Y 72.248,Z 441.483,A -85,B 0,C 180,E1 -28302.916,E2 -28302.916} C_VEL
LIN {X 0,Y 72.3,Z 441.445,A -85,B 0,C 180,E1 -28311.045,E2 -28311.045} C_VEL
LIN {X 0,Y 72.353,Z 441.518,A -85,B 0,C 180,E1 -28319.239,E2 -28319.239} C_VEL
LIN {X 0,Y 73.318,Z 444.129,A -85,B 0,C 180,E1 -28321.359,E2 -28321.359} C_VEL
LIN {X 0,Y 75.645,Z 447.195,A -85,B 0,C 180,E1 -28324.935,E2 -28324.935} C_VEL
LIN {X 0,Y 79.955,Z 454.385,A -85,B 0,C 180,E1 -28331.382,E2 -28331.382} C_VEL
LIN {X 0,Y 83.213,Z 461.141,A -85,B 0,C 180,E1 -28336.35,E2 -28336.35} C_VEL
LIN {X 0,Y 86.001,Z 468.264,A -85,B 0,C 180,E1 -28340.988,E2 -28340.988} C_VEL
LIN {X 0,Y 86.995,Z 473.532,A -85,B 0,C 180,E1 -28343.936,E2 -28343.936} C_VEL
LIN {X 0,Y 86.969,Z 481.616,A -85,B 0,C 180,E1 -28348.079,E2 -28348.079} C_VEL
LIN {X 0,Y 86.76,Z 486.116,A -85,B 0,C 180,E1 -28350.529,E2 -28350.529} C_VEL
LIN {X 0,Y 84.7,Z 491.079,A -85,B 0,C 180,E1 -28352.847,E2 -28352.847} C_VEL
LIN {X 0,Y 82.111,Z 495.437,A -85,B 0,C 180,E1 -28354.925,E2 -28354.925} C_VEL
LIN {X 0,Y 76.302,Z 501.989,A -85,B 0,C 180,E1 -28358.285,E2 -28358.285} C_VEL
LIN {X 0,Y 70.49,Z 508.078,A -85,B 0,C 180,E1 -28362.489,E2 -28362.489} C_VEL
LIN {X 0,Y 68.027,Z 511.607,A -85,B 0,C 180,E1 -28365.848,E2 -28365.848} C_VEL
LIN {X 0,Y 65.042,Z 518.174,A -85,B 0,C 180,E1 -28373.899,E2 -28373.899} C_VEL
LIN {X 0,Y 63.372,Z 522.627,A -85,B 0,C 180,E1 -28380.92,E2 -28380.92} C_VEL
LIN {X 0,Y 62.222,Z 527.26,A -85,B 0,C 180,E1 -28390.084,E2 -28390.084} C_VEL
LIN {X 0,Y 62.721,Z 531.702,A -85,B 0,C 180,E1 -28401.657,E2 -28401.657} C_VEL
LIN {X 0,Y 64.689,Z 534.239,A -85,B 0,C 180,E1 -28410.353,E2 -28410.353} C_VEL
LIN {X 0,Y 67.981,Z 536.057,A -85,B 0,C 180,E1 -28418.496,E2 -28418.496} C_VEL
LIN {X 0,Y 75.11,Z 537.381,A -85,B 0,C 180,E1 -28429.214,E2 -28429.214} C_VEL
LIN {X 0,Y 84.391,Z 537.121,A -85,B 0,C 180,E1 -28437.871,E2 -28437.871} C_VEL
LIN {X 0,Y 94.515,Z 535.356,A -85,B 0,C 180,E1 -28444.265,E2 -28444.265} C_VEL
LIN {X 0,Y 102.174,Z 533.289,A -85,B 0,C 180,E1 -28447.907,E2 -28447.907} C_VEL
LIN {X 0,Y 110.237,Z 530.418,A -85,B 0,C 180,E1 -28451.027,E2 -28451.027} C_VEL
LIN {X 0,Y 114.205,Z 528.741,A -85,B 0,C 180,E1 -28452.438,E2 -28452.438} C_VEL
LIN {X 0,Y 114.896,Z 528.38,A -85,B 0,C 180,E1 -28454.163,E2 -28454.163} C_VEL
LIN {X 0,Y 114.98,Z 528.305,A -85,B 0,C 180,E1 -28457.796,E2 -28457.796} C_VEL
LIN {X 0,Y 114.678,Z 528.633,A -85,B 0,C 180,E1 -28461.575,E2 -28461.575} C_VEL
LIN {X 0,Y 113.774,Z 529.513,A -85,B 0,C 180,E1 -28465.62,E2 -28465.62} C_VEL
LIN {X 0,Y 112.328,Z 530.654,A -85,B 0,C 180,E1 -28468.848,E2 -28468.848} C_VEL
LIN {X 0,Y 100.727,Z 535.327,A -85,B 0,C 180,E1 -28473.15,E2 -28473.15} C_VEL
LIN {X 0,Y 89.975,Z 538.436,A -85,B 0,C 180,E1 -28478.641,E2 -28478.641} C_VEL
LIN {X 0,Y 80.354,Z 540.176,A -85,B 0,C 180,E1 -28485.6,E2 -28485.6} C_VEL
LIN {X 0,Y 72.284,Z 540.571,A -85,B 0,C 180,E1 -28494.315,E2 -28494.315} C_VEL
LIN {X 0,Y 66.47,Z 539.576,A -85,B 0,C 180,E1 -28504.983,E2 -28504.983} C_VEL
LIN {X 0,Y 63.493,Z 537.188,A -85,B 0,C 180,E1 -28517.212,E2 -28517.212} C_VEL
LIN {X 0,Y 63.067,Z 534.4,A -85,B 0,C 180,E1 -28526.808,E2 -28526.808} C_VEL
LIN {X 0,Y 63.184,Z 533.277,A -85,B 0,C 180,E1 -28530.002,E2 -28530.002} C_VEL
LIN {X 0,Y 63.319,Z 528.934,A -85,B 0,C 180,E1 -28539.586,E2 -28539.586} C_VEL
LIN {X 0,Y 65.208,Z 522.267,A -85,B 0,C 180,E1 -28550.507,E2 -28550.507} C_VEL
LIN {X 0,Y 68.455,Z 515.012,A -85,B 0,C 180,E1 -28559.189,E2 -28559.189} C_VEL
LIN {X 0,Y 72.988,Z 505.962,A -85,B 0,C 180,E1 -28567.002,E2 -28567.002} C_VEL
LIN {X 0,Y 75.725,Z 500.59,A -85,B 0,C 180,E1 -28570.519,E2 -28570.519} C_VEL
LIN {X 0,Y 76.792,Z 496.313,A -85,B 0,C 180,E1 -28573.276,E2 -28573.276} C_VEL
LIN {X 0,Y 78.563,Z 485.777,A -85,B 0,C 180,E1 -28579.359,E2 -28579.359} C_VEL
LIN {X 0,Y 79.766,Z 475.642,A -85,B 0,C 180,E1 -28584.311,E2 -28584.311} C_VEL
LIN {X 0,Y 78.858,Z 469.803,A -85,B 0,C 180,E1 -28587.674,E2 -28587.674} C_VEL
LIN {X 0,Y 77.281,Z 463.77,A -85,B 0,C 180,E1 -28591.481,E2 -28591.481} C_VEL
LIN {X 0,Y 73.775,Z 456.411,A -85,B 0,C 180,E1 -28597.601,E2 -28597.601} C_VEL
LIN {X 0,Y 71.44,Z 452.021,A -85,B 0,C 180,E1 -28601.805,E2 -28601.805} C_VEL
LIN {X 0,Y 69.906,Z 450.004,A -85,B 0,C 180,E1 -28604.444,E2 -28604.444} C_VEL
LIN {X 0,Y 69.237,Z 448.367,A -85,B 0,C 180,E1 -28606.068,E2 -28606.068} C_VEL
LIN {X 0,Y 67.053,Z 445.433,A -85,B 0,C 180,E1 -28610.574,E2 -28610.574} C_VEL
LIN {X 0,Y 66.044,Z 442.948,A -85,B 0,C 180,E1 -28613.508,E2 -28613.508} C_VEL
LIN {X 0,Y 65.986,Z 442.257,A -85,B 0,C 180,E1 -28614.269,E2 -28614.269} C_VEL
LIN {X 0,Y 66.503,Z 442.198,A -85,B 0,C 180,E1 -28620,E2 -28620} C_VEL
LIN {X 0,Y 65.777,Z 442.274,A -85,B 0,C 180,E1 -28632.338,E2 -28632.338} C_VEL
LIN {X 0,Y 65.386,Z 442.286,A -85,B 0,C 180,E1 -28638.811,E2 -28638.811} C_VEL
LIN {X 0,Y 65.242,Z 442.354,A -85,B 0,C 180,E1 -28645.524,E2 -28645.524} C_VEL
LIN {X 0,Y 65.198,Z 442.327,A -85,B 0,C 180,E1 -28652.613,E2 -28652.613} C_VEL
LIN {X 0,Y 65.184,Z 442.351,A -85,B 0,C 180,E1 -28660.995,E2 -28660.995} C_VEL
LIN {X 0,Y 65.23,Z 442.492,A -85,B 0,C 180,E1 -28669.159,E2 -28669.159} C_VEL
LIN {X 0,Y 66.351,Z 445.359,A -85,B 0,C 180,E1 -28672.703,E2 -28672.703} C_VEL
LIN {X 0,Y 67.876,Z 447.006,A -85,B 0,C 180,E1 -28675.927,E2 -28675.927} C_VEL
LIN {X 0,Y 71.209,Z 452.029,A -85,B 0,C 180,E1 -28682.654,E2 -28682.654} C_VEL
LIN {X 0,Y 75.488,Z 459.806,A -85,B 0,C 180,E1 -28690.372,E2 -28690.372} C_VEL
LIN {X 0,Y 78.153,Z 466.058,A -85,B 0,C 180,E1 -28695.448,E2 -28695.448} C_VEL
LIN {X 0,Y 80.286,Z 472.216,A -85,B 0,C 180,E1 -28699.915,E2 -28699.915} C_VEL
LIN {X 0,Y 80.844,Z 476.666,A -85,B 0,C 180,E1 -28702.604,E2 -28702.604} C_VEL
LIN {X 0,Y 80.409,Z 485.29,A -85,B 0,C 180,E1 -28707.493,E2 -28707.493} C_VEL
LIN {X 0,Y 80.174,Z 487.39,A -85,B 0,C 180,E1 -28708.742,E2 -28708.742} C_VEL
LIN {X 0,Y 75.073,Z 497.682,A -85,B 0,C 180,E1 -28714.269,E2 -28714.269} C_VEL
LIN {X 0,Y 70.214,Z 507.217,A -85,B 0,C 180,E1 -28721.546,E2 -28721.546} C_VEL
LIN {X 0,Y 68.027,Z 511.607,A -85,B 0,C 180,E1 -28725.848,E2 -28725.848} C_VEL
LIN {X 0,Y 65.739,Z 514.969,A -85,B 0,C 180,E1 -28729.523,E2 -28729.523} C_VEL
LIN {X 0,Y 60.761,Z 519.783,A -85,B 0,C 180,E1 -28735.965,E2 -28735.965} C_VEL
LIN {X 0,Y 57.089,Z 523.197,A -85,B 0,C 180,E1 -28742.056,E2 -28742.056} C_VEL
LIN {X 0,Y 55.419,Z 525.662,A -85,B 0,C 180,E1 -28747.341,E2 -28747.341} C_VEL
LIN {X 0,Y 55.193,Z 526.469,A -85,B 0,C 180,E1 -28749.208,E2 -28749.208} C_VEL
LIN {X 0,Y 55.476,Z 530.679,A -85,B 0,C 180,E1 -28760.697,E2 -28760.697} C_VEL
LIN {X 0,Y 57.448,Z 533.571,A -85,B 0,C 180,E1 -28770.703,E2 -28770.703} C_VEL
LIN {X 0,Y 60.833,Z 535.667,A -85,B 0,C 180,E1 -28779.722,E2 -28779.722} C_VEL
LIN {X 0,Y 65.482,Z 537.054,A -85,B 0,C 180,E1 -28787.605,E2 -28787.605} C_VEL
LIN {X 0,Y 71.085,Z 537.699,A -85,B 0,C 180,E1 -28794.326,E2 -28794.326} C_VEL
LIN {X 0,Y 77.504,Z 537.714,A -85,B 0,C 180,E1 -28800,E2 -28800} C_VEL
LIN {X 0,Y 88.439,Z 536.432,A -85,B 0,C 180,E1 -28806.846,E2 -28806.846} C_VEL
LIN {X 0,Y 100.638,Z 533.537,A -85,B 0,C 180,E1 -28812.136,E2 -28812.136} C_VEL
LIN {X 0,Y 104.801,Z 532.231,A -85,B 0,C 180,E1 -28813.595,E2 -28813.595} C_VEL
LIN {X 0,Y 108.28,Z 530.977,A -85,B 0,C 180,E1 -28815.048,E2 -28815.048} C_VEL
LIN {X 0,Y 108.235,Z 531.062,A -85,B 0,C 180,E1 -28818.946,E2 -28818.946} C_VEL
LIN {X 0,Y 107.503,Z 531.706,A -85,B 0,C 180,E1 -28823.763,E2 -28823.763} C_VEL
LIN {X 0,Y 106.086,Z 532.561,A -85,B 0,C 180,E1 -28826.579,E2 -28826.579} C_VEL
LIN {X 0,Y 97.039,Z 535.663,A -85,B 0,C 180,E1 -28829.65,E2 -28829.65} C_VEL
LIN {X 0,Y 85.719,Z 538.543,A -85,B 0,C 180,E1 -28834.93,E2 -28834.93} C_VEL
LIN {X 0,Y 75.443,Z 540.046,A -85,B 0,C 180,E1 -28841.823,E2 -28841.823} C_VEL
LIN {X 0,Y 66.632,Z 540.16,A -85,B 0,C 180,E1 -28850.743,E2 -28850.743} C_VEL
LIN {X 0,Y 60.107,Z 538.944,A -85,B 0,C 180,E1 -28862.118,E2 -28862.118} C_VEL
LIN {X 0,Y 56.624,Z 536.38,A -85,B 0,C 180,E1 -28875.63,E2 -28875.63} C_VEL
LIN {X 0,Y 56.072,Z 533.407,A -85,B 0,C 180,E1 -28886.41,E2 -28886.41} C_VEL
LIN {X 0,Y 56.151,Z 532.182,A -85,B 0,C 180,E1 -28890.003,E2 -28890.003} C_VEL
LIN {X 0,Y 56.354,Z 527.613,A -85,B 0,C 180,E1 -28900.784,E2 -28900.784} C_VEL
LIN {X 0,Y 58.649,Z 520.696,A -85,B 0,C 180,E1 -28912.923,E2 -28912.923} C_VEL
LIN {X 0,Y 62.347,Z 513.13,A -85,B 0,C 180,E1 -28922.376,E2 -28922.376} C_VEL
LIN {X 0,Y 67.454,Z 503.695,A -85,B 0,C 180,E1 -28930.634,E2 -28930.634} C_VEL
LIN {X 0,Y 69.776,Z 499.02,A -85,B 0,C 180,E1 -28933.829,E2 -28933.829} C_VEL
LIN {X 0,Y 71.832,Z 488.998,A -85,B 0,C 180,E1 -28940.461,E2 -28940.461} C_VEL
LIN {X 0,Y 73.555,Z 478.797,A -85,B 0,C 180,E1 -28946.059,E2 -28946.059} C_VEL
LIN {X 0,Y 73.629,Z 476.203,A -85,B 0,C 180,E1 -28947.528,E2 -28947.528} C_VEL
LIN {X 0,Y 72.347,Z 468.978,A -85,B 0,C 180,E1 -28952.52,E2 -28952.52} C_VEL
LIN {X 0,Y 69.93,Z 463.075,A -85,B 0,C 180,E1 -28957.797,E2 -28957.797} C_VEL
LIN {X 0,Y 67.246,Z 457.347,A -85,B 0,C 180,E1 -28963.812,E2 -28963.812} C_VEL
LIN {X 0,Y 65.149,Z 453.243,A -85,B 0,C 180,E1 -28969.119,E2 -28969.119} C_VEL
LIN {X 0,Y 63.372,Z 450.622,A -85,B 0,C 180,E1 -28973.632,E2 -28973.632} C_VEL
LIN {X 0,Y 62.566,Z 448.384,A -85,B 0,C 180,E1 -28976.78,E2 -28976.78} C_VEL
LIN {X 0,Y 60.771,Z 446.818,A -85,B 0,C 180,E1 -28982.485,E2 -28982.485} C_VEL
LIN {X 0,Y 58.72,Z 443.849,A -85,B 0,C 180,E1 -28995.205,E2 -28995.205} C_VEL
LIN {X 0,Y 58.392,Z 444.273,A -85,B 0,C 180,E1 -29006.83,E2 -29006.83} C_VEL
LIN {X 0,Y 58.835,Z 445.585,A -85,B 0,C 180,E1 -29013.259,E2 -29013.259} C_VEL
LIN {X 0,Y 62.138,Z 448.868,A -85,B 0,C 180,E1 -29027.262,E2 -29027.262} C_VEL
LIN {X 0,Y 63.146,Z 451.446,A -85,B 0,C 180,E1 -29031.176,E2 -29031.176} C_VEL
LIN {X 0,Y 64.958,Z 453.814,A -85,B 0,C 180,E1 -29035.752,E2 -29035.752} C_VEL
LIN {X 0,Y 67.114,Z 457.53,A -85,B 0,C 180,E1 -29041.053,E2 -29041.053} C_VEL
LIN {X 0,Y 70.224,Z 463.81,A -85,B 0,C 180,E1 -29048.09,E2 -29048.09} C_VEL
LIN {X 0,Y 72.386,Z 469.184,A -85,B 0,C 180,E1 -29053.064,E2 -29053.064} C_VEL
LIN {X 0,Y 74.395,Z 475.563,A -85,B 0,C 180,E1 -29058.336,E2 -29058.336} C_VEL
LIN {X 0,Y 74.647,Z 479.149,A -85,B 0,C 180,E1 -29060.748,E2 -29060.748} C_VEL
LIN {X 0,Y 73.922,Z 487.312,A -85,B 0,C 180,E1 -29065.909,E2 -29065.909} C_VEL
LIN {X 0,Y 70.28,Z 494.739,A -85,B 0,C 180,E1 -29069.998,E2 -29069.998} C_VEL
LIN {X 0,Y 64.768,Z 504.844,A -85,B 0,C 180,E1 -29077.406,E2 -29077.406} C_VEL
LIN {X 0,Y 60.749,Z 512.289,A -85,B 0,C 180,E1 -29085.077,E2 -29085.077} C_VEL
LIN {X 0,Y 57.44,Z 519.393,A -85,B 0,C 180,E1 -29095.141,E2 -29095.141} C_VEL
LIN {X 0,Y 55.375,Z 525.535,A -85,B 0,C 180,E1 -29107.071,E2 -29107.071} C_VEL
LIN {X 0,Y 55.193,Z 526.469,A -85,B 0,C 180,E1 -29109.208,E2 -29109.208} C_VEL
LIN {X 0,Y 54.394,Z 528.714,A -85,B 0,C 180,E1 -29114.86,E2 -29114.86} C_VEL
LIN {X 0,Y 52.443,Z 531.68,A -85,B 0,C 180,E1 -29124.807,E2 -29124.807} C_VEL
LIN {X 0,Y 51.932,Z 533.551,A -85,B 0,C 180,E1 -29133.321,E2 -29133.321} C_VEL
LIN {X 0,Y 53.052,Z 534.798,A -85,B 0,C 180,E1 -29139.556,E2 -29139.556} C_VEL
LIN {X 0,Y 53.805,Z 535.166,A -85,B 0,C 180,E1 -29141.479,E2 -29141.479} C_VEL
LIN {X 0,Y 61.273,Z 537.371,A -85,B 0,C 180,E1 -29153.414,E2 -29153.414} C_VEL
LIN {X 0,Y 70.329,Z 538.105,A -85,B 0,C 180,E1 -29162.212,E2 -29162.212} C_VEL
LIN {X 0,Y 77.938,Z 537.833,A -85,B 0,C 180,E1 -29167.307,E2 -29167.307} C_VEL
LIN {X 0,Y 86.041,Z 536.841,A -85,B 0,C 180,E1 -29171.435,E2 -29171.435} C_VEL
LIN {X 0,Y 94.475,Z 535.182,A -85,B 0,C 180,E1 -29174.752,E2 -29174.752} C_VEL
LIN {X 0,Y 101.478,Z 533.287,A -85,B 0,C 180,E1 -29177.118,E2 -29177.118} C_VEL
LIN {X 0,Y 101.242,Z 533.491,A -85,B 0,C 180,E1 -29180.31,E2 -29180.31} C_VEL
LIN {X 0,Y 99.952,Z 534.19,A -85,B 0,C 180,E1 -29183.929,E2 -29183.929} C_VEL
LIN {X 0,Y 87.685,Z 537.498,A -85,B 0,C 180,E1 -29188.162,E2 -29188.162} C_VEL
LIN {X 0,Y 76.229,Z 539.381,A -85,B 0,C 180,E1 -29193.93,E2 -29193.93} C_VEL
LIN {X 0,Y 65.855,Z 539.94,A -85,B 0,C 180,E1 -29201.669,E2 -29201.669} C_VEL
LIN {X 0,Y 57.23,Z 539.183,A -85,B 0,C 180,E1 -29212.123,E2 -29212.123} C_VEL
LIN {X 0,Y 51.506,Z 537.065,A -85,B 0,C 180,E1 -29225.84,E2 -29225.84} C_VEL
LIN {X 0,Y 49.139,Z 533.475,A -85,B 0,C 180,E1 -29241.78,E2 -29241.78} C_VEL
LIN {X 0,Y 49.101,Z 531.056,A -85,B 0,C 180,E1 -29250.003,E2 -29250.003} C_VEL
LIN {X 0,Y 49.43,Z 526.283,A -85,B 0,C 180,E1 -29262.317,E2 -29262.317} C_VEL
LIN {X 0,Y 51.629,Z 520.201,A -85,B 0,C 180,E1 -29274.106,E2 -29274.106} C_VEL
LIN {X 0,Y 55.668,Z 512.581,A -85,B 0,C 180,E1 -29284.622,E2 -29284.622} C_VEL
LIN {X 0,Y 61.188,Z 503.093,A -85,B 0,C 180,E1 -29293.566,E2 -29293.566} C_VEL
LIN {X 0,Y 63.25,Z 499.38,A -85,B 0,C 180,E1 -29296.243,E2 -29296.243} C_VEL
LIN {X 0,Y 65.668,Z 489.575,A -85,B 0,C 180,E1 -29303.39,E2 -29303.39} C_VEL
LIN {X 0,Y 67.775,Z 479.528,A -85,B 0,C 180,E1 -29309.449,E2 -29309.449} C_VEL
LIN {X 0,Y 67.075,Z 473.636,A -85,B 0,C 180,E1 -29313.975,E2 -29313.975} C_VEL
LIN {X 0,Y 65.761,Z 469.326,A -85,B 0,C 180,E1 -29318.034,E2 -29318.034} C_VEL
LIN {X 0,Y 63.314,Z 463.268,A -85,B 0,C 180,E1 -29324.986,E2 -29324.986} C_VEL
LIN {X 0,Y 61.716,Z 459.662,A -85,B 0,C 180,E1 -29329.975,E2 -29329.975} C_VEL
LIN {X 0,Y 59.076,Z 454.094,A -85,B 0,C 180,E1 -29340,E2 -29340} C_VEL
LIN {X 0,Y 56.63,Z 450.826,A -85,B 0,C 180,E1 -29354.371,E2 -29354.371} C_VEL
LIN {X 0,Y 56.204,Z 450.718,A -85,B 0,C 180,E1 -29362.032,E2 -29362.032} C_VEL
LIN {X 0,Y 56.343,Z 451.578,A -85,B 0,C 180,E1 -29369.93,E2 -29369.93} C_VEL
LIN {X 0,Y 58.981,Z 455.167,A -85,B 0,C 180,E1 -29385.638,E2 -29385.638} C_VEL
LIN {X 0,Y 59.785,Z 457.5,A -85,B 0,C 180,E1 -29389.762,E2 -29389.762} C_VEL
LIN {X 0,Y 61.476,Z 460.226,A -85,B 0,C 180,E1 -29395.135,E2 -29395.135} C_VEL
LIN {X 0,Y 63.694,Z 464.989,A -85,B 0,C 180,E1 -29401.972,E2 -29401.972} C_VEL
LIN {X 0,Y 65.793,Z 469.769,A -85,B 0,C 180,E1 -29407.793,E2 -29407.793} C_VEL
LIN {X 0,Y 67.894,Z 476.389,A -85,B 0,C 180,E1 -29414.328,E2 -29414.328} C_VEL
LIN {X 0,Y 68.592,Z 479.831,A -85,B 0,C 180,E1 -29417.334,E2 -29417.334} C_VEL
LIN {X 0,Y 67.8,Z 487.237,A -85,B 0,C 180,E1 -29422.553,E2 -29422.553} C_VEL
LIN {X 0,Y 67.638,Z 488.274,A -85,B 0,C 180,E1 -29423.285,E2 -29423.285} C_VEL
